# B&R Automation Studio project AAU12Segmenter (part 3)

```iecst
	(*________________________________________*)
	(*_____________KUKA5 Mappings_____________*)
	(*________________________________________*)

	::InputVariables[4,0] AT %IB."KUKA5_KRC4_ProfiNet_5_0".Module001_8_digital_inputs_I_00;
	::InputVariables[4,1] AT %IB."KUKA5_KRC4_ProfiNet_5_0".Module001_8_digital_inputs_I_01;
	::InputVariables[4,2] AT %IB."KUKA5_KRC4_ProfiNet_5_0".Module001_8_digital_inputs_I_02;
	::InputVariables[4,3] AT %IB."KUKA5_KRC4_ProfiNet_5_0".Module001_8_digital_inputs_I_03;
	::InputVariables[4,4] AT %IB."KUKA5_KRC4_ProfiNet_5_0".Module001_8_digital_inputs_I_04;
	::InputVariables[4,5] AT %IB."KUKA5_KRC4_ProfiNet_5_0".Module001_8_digital_inputs_I_05;
	::InputVariables[4,6] AT %IB."KUKA5_KRC4_ProfiNet_5_0".Module001_8_digital_inputs_I_06;
	::InputVariables[4,7] AT %IB."KUKA5_KRC4_ProfiNet_5_0".Module001_8_digital_inputs_I_07;
	::InputVariables[4,8] AT %IB."KUKA5_KRC4_ProfiNet_5_0".Module001_8_digital_inputs_I_08;
	::InputVariables[4,9] AT %IB."KUKA5_KRC4_ProfiNet_5_0".Module001_8_digital_inputs_I_09;
	::InputVariables[4,10] AT %IB."KUKA5_KRC4_ProfiNet_5_0".Module001_8_digital_inputs_I_10;
	::InputVariables[4,11] AT %IB."KUKA5_KRC4_ProfiNet_5_0".Module001_8_digital_inputs_I_11;
	::InputVariables[4,12] AT %IB."KUKA5_KRC4_ProfiNet_5_0".Module001_8_digital_inputs_I_12;
	::InputVariables[4,13] AT %IB."KUKA5_KRC4_ProfiNet_5_0".Module001_8_digital_inputs_I_13;
	::InputVariables[4,14] AT %IB."KUKA5_KRC4_ProfiNet_5_0".Module001_8_digital_inputs_I_14;
	::InputVariables[4,15] AT %IB."KUKA5_KRC4_ProfiNet_5_0".Module001_8_digital_inputs_I_15;
	::InputVariables[4,16] AT %IB."KUKA5_KRC4_ProfiNet_5_0".Module001_8_digital_inputs_I_16;
	::InputVariables[4,17] AT %IB."KUKA5_KRC4_ProfiNet_5_0".Module001_8_digital_inputs_I_17;
	::InputVariables[4,18] AT %IB."KUKA5_KRC4_ProfiNet_5_0".Module001_8_digital_inputs_I_18;
	::InputVariables[4,19] AT %IB."KUKA5_KRC4_ProfiNet_5_0".Module001_8_digital_inputs_I_19;
	::InputVariables[4,20] AT %IB."KUKA5_KRC4_ProfiNet_5_0".Module001_8_digital_inputs_I_20;
	::InputVariables[4,21] AT %IB."KUKA5_KRC4_ProfiNet_5_0".Module001_8_digital_inputs_I_21;
	::InputVariables[4,22] AT %IB."KUKA5_KRC4_ProfiNet_5_0".Module001_8_digital_inputs_I_22;
	::InputVariables[4,23] AT %IB."KUKA5_KRC4_ProfiNet_5_0".Module001_8_digital_inputs_I_23;
	::InputVariables[4,24] AT %IB."KUKA5_KRC4_ProfiNet_5_0".Module001_8_digital_inputs_I_24;
	::InputVariables[4,25] AT %IB."KUKA5_KRC4_ProfiNet_5_0".Module001_8_digital_inputs_I_25;
	::InputVariables[4,26] AT %IB."KUKA5_KRC4_ProfiNet_5_0".Module001_8_digital_inputs_I_26;
	::InputVariables[4,27] AT %IB."KUKA5_KRC4_ProfiNet_5_0".Module001_8_digital_inputs_I_27;
	::InputVariables[4,28] AT %IB."KUKA5_KRC4_ProfiNet_5_0".Module001_8_digital_inputs_I_28;
	::InputVariables[4,29] AT %IB."KUKA5_KRC4_ProfiNet_5_0".Module001_8_digital_inputs_I_29;
	::InputVariables[4,30] AT %IB."KUKA5_KRC4_ProfiNet_5_0".Module001_8_digital_inputs_I_30;
	::InputVariables[4,31] AT %IB."KUKA5_KRC4_ProfiNet_5_0".Module001_8_digital_inputs_I_31;
	::InputVariables[4,32] AT %IB."KUKA5_KRC4_ProfiNet_5_0".Module001_8_digital_inputs_I_32;
	::InputVariables[4,33] AT %IB."KUKA5_KRC4_ProfiNet_5_0".Module001_8_digital_inputs_I_33;
	::InputVariables[4,34] AT %IB."KUKA5_KRC4_ProfiNet_5_0".Module001_8_digital_inputs_I_34;
	::InputVariables[4,35] AT %IB."KUKA5_KRC4_ProfiNet_5_0".Module001_8_digital_inputs_I_35;
	::InputVariables[4,36] AT %IB."KUKA5_KRC4_ProfiNet_5_0".Module001_8_digital_inputs_I_36;
	::InputVariables[4,37] AT %IB."KUKA5_KRC4_ProfiNet_5_0".Module001_8_digital_inputs_I_37;
	::InputVariables[4,38] AT %IB."KUKA5_KRC4_ProfiNet_5_0".Module001_8_digital_inputs_I_38;
	::InputVariables[4,39] AT %IB."KUKA5_KRC4_ProfiNet_5_0".Module001_8_digital_inputs_I_39;
	::InputVariables[4,40] AT %IB."KUKA5_KRC4_ProfiNet_5_0".Module001_8_digital_inputs_I_40;
	::InputVariables[4,41] AT %IB."KUKA5_KRC4_ProfiNet_5_0".Module001_8_digital_inputs_I_41;
	::InputVariables[4,42] AT %IB."KUKA5_KRC4_ProfiNet_5_0".Module001_8_digital_inputs_I_42;
	::InputVariables[4,43] AT %IB."KUKA5_KRC4_ProfiNet_5_0".Module001_8_digital_inputs_I_43;
	::InputVariables[4,44] AT %IB."KUKA5_KRC4_ProfiNet_5_0".Module001_8_digital_inputs_I_44;
	::InputVariables[4,45] AT %IB."KUKA5_KRC4_ProfiNet_5_0".Module001_8_digital_inputs_I_45;
	::InputVariables[4,46] AT %IB."KUKA5_KRC4_ProfiNet_5_0".Module001_8_digital_inputs_I_46;
	::InputVariables[4,47] AT %IB."KUKA5_KRC4_ProfiNet_5_0".Module001_8_digital_inputs_I_47;
	::InputVariables[4,48] AT %IB."KUKA5_KRC4_ProfiNet_5_0".Module001_8_digital_inputs_I_48;
	::InputVariables[4,49] AT %IB."KUKA5_KRC4_ProfiNet_5_0".Module001_8_digital_inputs_I_49;
	::InputVariables[4,50] AT %IB."KUKA5_KRC4_ProfiNet_5_0".Module001_8_digital_inputs_I_50;
	::InputVariables[4,51] AT %IB."KUKA5_KRC4_ProfiNet_5_0".Module001_8_digital_inputs_I_51;
	::InputVariables[4,52] AT %IB."KUKA5_KRC4_ProfiNet_5_0".Module001_8_digital_inputs_I_52;
	::InputVariables[4,53] AT %IB."KUKA5_KRC4_ProfiNet_5_0".Module001_8_digital_inputs_I_53;
	::InputVariables[4,54] AT %IB."KUKA5_KRC4_ProfiNet_5_0".Module001_8_digital_inputs_I_54;
	::InputVariables[4,55] AT %IB."KUKA5_KRC4_ProfiNet_5_0".Module001_8_digital_inputs_I_55;
	::InputVariables[4,56] AT %IB."KUKA5_KRC4_ProfiNet_5_0".Module001_8_digital_inputs_I_56;
	::InputVariables[4,57] AT %IB."KUKA5_KRC4_ProfiNet_5_0".Module001_8_digital_inputs_I_57;
	::InputVariables[4,58] AT %IB."KUKA5_KRC4_ProfiNet_5_0".Module001_8_digital_inputs_I_58;
	::InputVariables[4,59] AT %IB."KUKA5_KRC4_ProfiNet_5_0".Module001_8_digital_inputs_I_59;
	::InputVariables[4,60] AT %IB."KUKA5_KRC4_ProfiNet_5_0".Module001_8_digital_inputs_I_60;
	::InputVariables[4,61] AT %IB."KUKA5_KRC4_ProfiNet_5_0".Module001_8_digital_inputs_I_61;
	::InputVariables[4,62] AT %IB."KUKA5_KRC4_ProfiNet_5_0".Module001_8_digital_inputs_I_62;
	::InputVariables[4,63] AT %IB."KUKA5_KRC4_ProfiNet_5_0".Module001_8_digital_inputs_I_63;
	::InputVariables[4,64] AT %IB."KUKA5_KRC4_ProfiNet_5_0".Module001_8_digital_inputs_I_64;
	::InputVariables[4,65] AT %IB."KUKA5_KRC4_ProfiNet_5_0".Module001_8_digital_inputs_I_65;
	::InputVariables[4,66] AT %IB."KUKA5_KRC4_ProfiNet_5_0".Module001_8_digital_inputs_I_66;
	::InputVariables[4,67] AT %IB."KUKA5_KRC4_ProfiNet_5_0".Module001_8_digital_inputs_I_67;
	::InputVariables[4,68] AT %IB."KUKA5_KRC4_ProfiNet_5_0".Module001_8_digital_inputs_I_68;
	::InputVariables[4,69] AT %IB."KUKA5_KRC4_ProfiNet_5_0".Module001_8_digital_inputs_I_69;
	::InputVariables[4,70] AT %IB."KUKA5_KRC4_ProfiNet_5_0".Module001_8_digital_inputs_I_70;
	::InputVariables[4,71] AT %IB."KUKA5_KRC4_ProfiNet_5_0".Module001_8_digital_inputs_I_71;
	::InputVariables[4,72] AT %IB."KUKA5_KRC4_ProfiNet_5_0".Module001_8_digital_inputs_I_72;
	::InputVariables[4,73] AT %IB."KUKA5_KRC4_ProfiNet_5_0".Module001_8_digital_inputs_I_73;
	::InputVariables[4,74] AT %IB."KUKA5_KRC4_ProfiNet_5_0".Module001_8_digital_inputs_I_74;
	::InputVariables[4,75] AT %IB."KUKA5_KRC4_ProfiNet_5_0".Module001_8_digital_inputs_I_75;
	::InputVariables[4,76] AT %IB."KUKA5_KRC4_ProfiNet_5_0".Module001_8_digital_inputs_I_76;
	::InputVariables[4,77] AT %IB."KUKA5_KRC4_ProfiNet_5_0".Module001_8_digital_inputs_I_77;
	::InputVariables[4,78] AT %IB."KUKA5_KRC4_ProfiNet_5_0".Module001_8_digital_inputs_I_78;
	::InputVariables[4,79] AT %IB."KUKA5_KRC4_ProfiNet_5_0".Module001_8_digital_inputs_I_79;
	::InputVariables[4,80] AT %IB."KUKA5_KRC4_ProfiNet_5_0".Module001_8_digital_inputs_I_80;
	::InputVariables[4,81] AT %IB."KUKA5_KRC4_ProfiNet_5_0".Module001_8_digital_inputs_I_81;
	::InputVariables[4,82] AT %IB."KUKA5_KRC4_ProfiNet_5_0".Module001_8_digital_inputs_I_82;
	::InputVariables[4,83] AT %IB."KUKA5_KRC4_ProfiNet_5_0".Module001_8_digital_inputs_I_83;
	::InputVariables[4,84] AT %IB."KUKA5_KRC4_ProfiNet_5_0".Module001_8_digital_inputs_I_84;
	::InputVariables[4,85] AT %IB."KUKA5_KRC4_ProfiNet_5_0".Module001_8_digital_inputs_I_85;
	::InputVariables[4,86] AT %IB."KUKA5_KRC4_ProfiNet_5_0".Module001_8_digital_inputs_I_86;
	::InputVariables[4,87] AT %IB."KUKA5_KRC4_ProfiNet_5_0".Module001_8_digital_inputs_I_87;
	::InputVariables[4,88] AT %IB."KUKA5_KRC4_ProfiNet_5_0".Module001_8_digital_inputs_I_88;
	::InputVariables[4,89] AT %IB."KUKA5_KRC4_ProfiNet_5_0".Module001_8_digital_inputs_I_89;
	::InputVariables[4,90] AT %IB."KUKA5_KRC4_ProfiNet_5_0".Module001_8_digital_inputs_I_90;
	::InputVariables[4,91] AT %IB."KUKA5_KRC4_ProfiNet_5_0".Module001_8_digital_inputs_I_91;
	::InputVariables[4,92] AT %IB."KUKA5_KRC4_ProfiNet_5_0".Module001_8_digital_inputs_I_92;
	::InputVariables[4,93] AT %IB."KUKA5_KRC4_ProfiNet_5_0".Module001_8_digital_inputs_I_93;
	::InputVariables[4,94] AT %IB."KUKA5_KRC4_ProfiNet_5_0".Module001_8_digital_inputs_I_94;
	::InputVariables[4,95] AT %IB."KUKA5_KRC4_ProfiNet_5_0".Module001_8_digital_inputs_I_95;
	::InputVariables[4,96] AT %IB."KUKA5_KRC4_ProfiNet_5_0".Module001_8_digital_inputs_I_96;
	::InputVariables[4,97] AT %IB."KUKA5_KRC4_ProfiNet_5_0".Module001_8_digital_inputs_I_97;
	::InputVariables[4,98] AT %IB."KUKA5_KRC4_ProfiNet_5_0".Module001_8_digital_inputs_I_98;
	::InputVariables[4,99] AT %IB."KUKA5_KRC4_ProfiNet_5_0".Module001_8_digital_inputs_I_99;
	::InputVariables[4,100] AT %IB."KUKA5_KRC4_ProfiNet_5_0".Module001_8_digital_inputs_I_100;
	::InputVariables[4,101] AT %IB."KUKA5_KRC4_ProfiNet_5_0".Module001_8_digital_inputs_I_101;
	::InputVariables[4,102] AT %IB."KUKA5_KRC4_ProfiNet_5_0".Module001_8_digital_inputs_I_102;
	::InputVariables[4,103] AT %IB."KUKA5_KRC4_ProfiNet_5_0".Module001_8_digital_inputs_I_103;
	::InputVariables[4,104] AT %IB."KUKA5_KRC4_ProfiNet_5_0".Module001_8_digital_inputs_I_104;
	::InputVariables[4,105] AT %IB."KUKA5_KRC4_ProfiNet_5_0".Module001_8_digital_inputs_I_105;
	::InputVariables[4,106] AT %IB."KUKA5_KRC4_ProfiNet_5_0".Module001_8_digital_inputs_I_106;
	::InputVariables[4,107] AT %IB."KUKA5_KRC4_ProfiNet_5_0".Module001_8_digital_inputs_I_107;
	::InputVariables[4,108] AT %IB."KUKA5_KRC4_ProfiNet_5_0".Module001_8_digital_inputs_I_108;
	::InputVariables[4,109] AT %IB."KUKA5_KRC4_ProfiNet_5_0".Module001_8_digital_inputs_I_109;
	::InputVariables[4,110] AT %IB."KUKA5_KRC4_ProfiNet_5_0".Module001_8_digital_inputs_I_110;
	::InputVariables[4,111] AT %IB."KUKA5_KRC4_ProfiNet_5_0".Module001_8_digital_inputs_I_111;
	::InputVariables[4,112] AT %IB."KUKA5_KRC4_ProfiNet_5_0".Module001_8_digital_inputs_I_112;
	::InputVariables[4,113] AT %IB."KUKA5_KRC4_ProfiNet_5_0".Module001_8_digital_inputs_I_113;
	::InputVariables[4,114] AT %IB."KUKA5_KRC4_ProfiNet_5_0".Module001_8_digital_inputs_I_114;
	::InputVariables[4,115] AT %IB."KUKA5_KRC4_ProfiNet_5_0".Module001_8_digital_inputs_I_115;
	::InputVariables[4,116] AT %IB."KUKA5_KRC4_ProfiNet_5_0".Module001_8_digital_inputs_I_116;
	::InputVariables[4,117] AT %IB."KUKA5_KRC4_ProfiNet_5_0".Module001_8_digital_inputs_I_117;
	::InputVariables[4,118] AT %IB."KUKA5_KRC4_ProfiNet_5_0".Module001_8_digital_inputs_I_118;
	::InputVariables[4,119] AT %IB."KUKA5_KRC4_ProfiNet_5_0".Module001_8_digital_inputs_I_119;
	::InputVariables[4,120] AT %IB."KUKA5_KRC4_ProfiNet_5_0".Module001_8_digital_inputs_I_120;
	::InputVariables[4,121] AT %IB."KUKA5_KRC4_ProfiNet_5_0".Module001_8_digital_inputs_I_121;
	::InputVariables[4,122] AT %IB."KUKA5_KRC4_ProfiNet_5_0".Module001_8_digital_inputs_I_122;
	::InputVariables[4,123] AT %IB."KUKA5_KRC4_ProfiNet_5_0".Module001_8_digital_inputs_I_123;
	::InputVariables[4,124] AT %IB."KUKA5_KRC4_ProfiNet_5_0".Module001_8_digital_inputs_I_124;
	::InputVariables[4,125] AT %IB."KUKA5_KRC4_ProfiNet_5_0".Module001_8_digital_inputs_I_125;
	::InputVariables[4,126] AT %IB."KUKA5_KRC4_ProfiNet_5_0".Module001_8_digital_inputs_I_126;
	::InputVariables[4,127] AT %IB."KUKA5_KRC4_ProfiNet_5_0".Module001_8_digital_inputs_I_127;
	::InputVariables[4,128] AT %IB."KUKA5_KRC4_ProfiNet_5_0".Module001_8_digital_inputs_I_128;
	::InputVariables[4,129] AT %IB."KUKA5_KRC4_ProfiNet_5_0".Module001_8_digital_inputs_I_129;
	::InputVariables[4,130] AT %IB."KUKA5_KRC4_ProfiNet_5_0".Module001_8_digital_inputs_I_130;
	::InputVariables[4,131] AT %IB."KUKA5_KRC4_ProfiNet_5_0".Module001_8_digital_inputs_I_131;
	::InputVariables[4,132] AT %IB."KUKA5_KRC4_ProfiNet_5_0".Module001_8_digital_inputs_I_132;
	::InputVariables[4,133] AT %IB."KUKA5_KRC4_ProfiNet_5_0".Module001_8_digital_inputs_I_133;
	::InputVariables[4,134] AT %IB."KUKA5_KRC4_ProfiNet_5_0".Module001_8_digital_inputs_I_134;
	::InputVariables[4,135] AT %IB."KUKA5_KRC4_ProfiNet_5_0".Module001_8_digital_inputs_I_135;
	::InputVariables[4,136] AT %IB."KUKA5_KRC4_ProfiNet_5_0".Module001_8_digital_inputs_I_136;
	::InputVariables[4,137] AT %IB."KUKA5_KRC4_ProfiNet_5_0".Module001_8_digital_inputs_I_137;
	::InputVariables[4,138] AT %IB."KUKA5_KRC4_ProfiNet_5_0".Module001_8_digital_inputs_I_138;
	::InputVariables[4,139] AT %IB."KUKA5_KRC4_ProfiNet_5_0".Module001_8_digital_inputs_I_139;
	::InputVariables[4,140] AT %IB."KUKA5_KRC4_ProfiNet_5_0".Module001_8_digital_inputs_I_140;
	::InputVariables[4,141] AT %IB."KUKA5_KRC4_ProfiNet_5_0".Module001_8_digital_inputs_I_141;
	::InputVariables[4,142] AT %IB."KUKA5_KRC4_ProfiNet_5_0".Module001_8_digital_inputs_I_142;
	::InputVariables[4,143] AT %IB."KUKA5_KRC4_ProfiNet_5_0".Module001_8_digital_inputs_I_143;
	::InputVariables[4,144] AT %IB."KUKA5_KRC4_ProfiNet_5_0".Module001_8_digital_inputs_I_144;
	::InputVariables[4,145] AT %IB."KUKA5_KRC4_ProfiNet_5_0".Module001_8_digital_inputs_I_145;
	::InputVariables[4,146] AT %IB."KUKA5_KRC4_ProfiNet_5_0".Module001_8_digital_inputs_I_146;
	::InputVariables[4,147] AT %IB."KUKA5_KRC4_ProfiNet_5_0".Module001_8_digital_inputs_I_147;
	::InputVariables[4,148] AT %IB."KUKA5_KRC4_ProfiNet_5_0".Module001_8_digital_inputs_I_148;
	::InputVariables[4,149] AT %IB."KUKA5_KRC4_ProfiNet_5_0".Module001_8_digital_inputs_I_149;
	::InputVariables[4,150] AT %IB."KUKA5_KRC4_ProfiNet_5_0".Module001_8_digital_inputs_I_150;
	::InputVariables[4,151] AT %IB."KUKA5_KRC4_ProfiNet_5_0".Module001_8_digital_inputs_I_151;
	::InputVariables[4,152] AT %IB."KUKA5_KRC4_ProfiNet_5_0".Module001_8_digital_inputs_I_152;
	::InputVariables[4,153] AT %IB."KUKA5_KRC4_ProfiNet_5_0".Module001_8_digital_inputs_I_153;
	::InputVariables[4,154] AT %IB."KUKA5_KRC4_ProfiNet_5_0".Module001_8_digital_inputs_I_154;
	::InputVariables[4,155] AT %IB."KUKA5_KRC4_ProfiNet_5_0".Module001_8_digital_inputs_I_155;
	::InputVariables[4,156] AT %IB."KUKA5_KRC4_ProfiNet_5_0".Module001_8_digital_inputs_I_156;
	::InputVariables[4,157] AT %IB."KUKA5_KRC4_ProfiNet_5_0".Module001_8_digital_inputs_I_157;
	::InputVariables[4,158] AT %IB."KUKA5_KRC4_ProfiNet_5_0".Module001_8_digital_inputs_I_158;
	::InputVariables[4,159] AT %IB."KUKA5_KRC4_ProfiNet_5_0".Module001_8_digital_inputs_I_159;
	::InputVariables[4,160] AT %IB."KUKA5_KRC4_ProfiNet_5_0".Module001_8_digital_inputs_I_160;
	::InputVariables[4,161] AT %IB."KUKA5_KRC4_ProfiNet_5_0".Module001_8_digital_inputs_I_161;
	::InputVariables[4,162] AT %IB."KUKA5_KRC4_ProfiNet_5_0".Module001_8_digital_inputs_I_162;
	::InputVariables[4,163] AT %IB."KUKA5_KRC4_ProfiNet_5_0".Module001_8_digital_inputs_I_163;
	::InputVariables[4,164] AT %IB."KUKA5_KRC4_ProfiNet_5_0".Module001_8_digital_inputs_I_164;
	::InputVariables[4,165] AT %IB."KUKA5_KRC4_ProfiNet_5_0".Module001_8_digital_inputs_I_165;
	::InputVariables[4,166] AT %IB."KUKA5_KRC4_ProfiNet_5_0".Module001_8_digital_inputs_I_166;
	::InputVariables[4,167] AT %IB."KUKA5_KRC4_ProfiNet_5_0".Module001_8_digital_inputs_I_167;
	::InputVariables[4,168] AT %IB."KUKA5_KRC4_ProfiNet_5_0".Module001_8_digital_inputs_I_168;
	::InputVariables[4,169] AT %IB."KUKA5_KRC4_ProfiNet_5_0".Module001_8_digital_inputs_I_169;
	::InputVariables[4,170] AT %IB."KUKA5_KRC4_ProfiNet_5_0".Module001_8_digital_inputs_I_170;
	::InputVariables[4,171] AT %IB."KUKA5_KRC4_ProfiNet_5_0".Module001_8_digital_inputs_I_171;
	::InputVariables[4,172] AT %IB."KUKA5_KRC4_ProfiNet_5_0".Module001_8_digital_inputs_I_172;
	::InputVariables[4,173] AT %IB."KUKA5_KRC4_ProfiNet_5_0".Module001_8_digital_inputs_I_173;
	::InputVariables[4,174] AT %IB."KUKA5_KRC4_ProfiNet_5_0".Module001_8_digital_inputs_I_174;
	::InputVariables[4,175] AT %IB."KUKA5_KRC4_ProfiNet_5_0".Module001_8_digital_inputs_I_175;
	::InputVariables[4,176] AT %IB."KUKA5_KRC4_ProfiNet_5_0".Module001_8_digital_inputs_I_176;
	::InputVariables[4,177] AT %IB."KUKA5_KRC4_ProfiNet_5_0".Module001_8_digital_inputs_I_177;
	::InputVariables[4,178] AT %IB."KUKA5_KRC4_ProfiNet_5_0".Module001_8_digital_inputs_I_178;
	::InputVariables[4,179] AT %IB."KUKA5_KRC4_ProfiNet_5_0".Module001_8_digital_inputs_I_179;
	::InputVariables[4,180] AT %IB."KUKA5_KRC4_ProfiNet_5_0".Module001_8_digital_inputs_I_180;
	::InputVariables[4,181] AT %IB."KUKA5_KRC4_ProfiNet_5_0".Module001_8_digital_inputs_I_181;
	::InputVariables[4,182] AT %IB."KUKA5_KRC4_ProfiNet_5_0".Module001_8_digital_inputs_I_182;
	::InputVariables[4,183] AT %IB."KUKA5_KRC4_ProfiNet_5_0".Module001_8_digital_inputs_I_183;
	::InputVariables[4,184] AT %IB."KUKA5_KRC4_ProfiNet_5_0".Module001_8_digital_inputs_I_184;
	::InputVariables[4,185] AT %IB."KUKA5_KRC4_ProfiNet_5_0".Module001_8_digital_inputs_I_185;
	::InputVariables[4,186] AT %IB."KUKA5_KRC4_ProfiNet_5_0".Module001_8_digital_inputs_I_186;
	::InputVariables[4,187] AT %IB."KUKA5_KRC4_ProfiNet_5_0".Module001_8_digital_inputs_I_187;
	::InputVariables[4,188] AT %IB."KUKA5_KRC4_ProfiNet_5_0".Module001_8_digital_inputs_I_188;
	::InputVariables[4,189] AT %IB."KUKA5_KRC4_ProfiNet_5_0".Module001_8_digital_inputs_I_189;
	::InputVariables[4,190] AT %IB."KUKA5_KRC4_ProfiNet_5_0".Module001_8_digital_inputs_I_190;
	::InputVariables[4,191] AT %IB."KUKA5_KRC4_ProfiNet_5_0".Module001_8_digital_inputs_I_191;
	::InputVariables[4,192] AT %IB."KUKA5_KRC4_ProfiNet_5_0".Module001_8_digital_inputs_I_192;
	::InputVariables[4,193] AT %IB."KUKA5_KRC4_ProfiNet_5_0".Module001_8_digital_inputs_I_193;
	::InputVariables[4,194] AT %IB."KUKA5_KRC4_ProfiNet_5_0".Module001_8_digital_inputs_I_194;
	::InputVariables[4,195] AT %IB."KUKA5_KRC4_ProfiNet_5_0".Module001_8_digital_inputs_I_195;
	::InputVariables[4,196] AT %IB."KUKA5_KRC4_ProfiNet_5_0".Module001_8_digital_inputs_I_196;
	::InputVariables[4,197] AT %IB."KUKA5_KRC4_ProfiNet_5_0".Module001_8_digital_inputs_I_197;
	::InputVariables[4,198] AT %IB."KUKA5_KRC4_ProfiNet_5_0".Module001_8_digital_inputs_I_198;
	::InputVariables[4,199] AT %IB."KUKA5_KRC4_ProfiNet_5_0".Module001_8_digital_inputs_I_199;
	::InputVariables[4,200] AT %IB."KUKA5_KRC4_ProfiNet_5_0".Module001_8_digital_inputs_I_200;
	::InputVariables[4,201] AT %IB."KUKA5_KRC4_ProfiNet_5_0".Module001_8_digital_inputs_I_201;
	::InputVariables[4,202] AT %IB."KUKA5_KRC4_ProfiNet_5_0".Module001_8_digital_inputs_I_202;
	::InputVariables[4,203] AT %IB."KUKA5_KRC4_ProfiNet_5_0".Module001_8_digital_inputs_I_203;
	::InputVariables[4,204] AT %IB."KUKA5_KRC4_ProfiNet_5_0".Module001_8_digital_inputs_I_204;
	::InputVariables[4,205] AT %IB."KUKA5_KRC4_ProfiNet_5_0".Module001_8_digital_inputs_I_205;
	::InputVariables[4,206] AT %IB."KUKA5_KRC4_ProfiNet_5_0".Module001_8_digital_inputs_I_206;
	::InputVariables[4,207] AT %IB."KUKA5_KRC4_ProfiNet_5_0".Module001_8_digital_inputs_I_207;
	::InputVariables[4,208] AT %IB."KUKA5_KRC4_ProfiNet_5_0".Module001_8_digital_inputs_I_208;
	::InputVariables[4,209] AT %IB."KUKA5_KRC4_ProfiNet_5_0".Module001_8_digital_inputs_I_209;
	::InputVariables[4,210] AT %IB."KUKA5_KRC4_ProfiNet_5_0".Module001_8_digital_inputs_I_210;
	::InputVariables[4,211] AT %IB."KUKA5_KRC4_ProfiNet_5_0".Module001_8_digital_inputs_I_211;
	::InputVariables[4,212] AT %IB."KUKA5_KRC4_ProfiNet_5_0".Module001_8_digital_inputs_I_212;
	::InputVariables[4,213] AT %IB."KUKA5_KRC4_ProfiNet_5_0".Module001_8_digital_inputs_I_213;
	::InputVariables[4,214] AT %IB."KUKA5_KRC4_ProfiNet_5_0".Module001_8_digital_inputs_I_214;
	::InputVariables[4,215] AT %IB."KUKA5_KRC4_ProfiNet_5_0".Module001_8_digital_inputs_I_215;
	::InputVariables[4,216] AT %IB."KUKA5_KRC4_ProfiNet_5_0".Module001_8_digital_inputs_I_216;
	::InputVariables[4,217] AT %IB."KUKA5_KRC4_ProfiNet_5_0".Module001_8_digital_inputs_I_217;
	::InputVariables[4,218] AT %IB."KUKA5_KRC4_ProfiNet_5_0".Module001_8_digital_inputs_I_218;
	::InputVariables[4,219] AT %IB."KUKA5_KRC4_ProfiNet_5_0".Module001_8_digital_inputs_I_219;
	::InputVariables[4,220] AT %IB."KUKA5_KRC4_ProfiNet_5_0".Module001_8_digital_inputs_I_220;
	::InputVariables[4,221] AT %IB."KUKA5_KRC4_ProfiNet_5_0".Module001_8_digital_inputs_I_221;
	::InputVariables[4,222] AT %IB."KUKA5_KRC4_ProfiNet_5_0".Module001_8_digital_inputs_I_222;
	::InputVariables[4,223] AT %IB."KUKA5_KRC4_ProfiNet_5_0".Module001_8_digital_inputs_I_223;
	::InputVariables[4,224] AT %IB."KUKA5_KRC4_ProfiNet_5_0".Module001_8_digital_inputs_I_224;
	::InputVariables[4,225] AT %IB."KUKA5_KRC4_ProfiNet_5_0".Module001_8_digital_inputs_I_225;
	::InputVariables[4,226] AT %IB."KUKA5_KRC4_ProfiNet_5_0".Module001_8_digital_inputs_I_226;
	::InputVariables[4,227] AT %IB."KUKA5_KRC4_ProfiNet_5_0".Module001_8_digital_inputs_I_227;
	::InputVariables[4,228] AT %IB."KUKA5_KRC4_ProfiNet_5_0".Module001_8_digital_inputs_I_228;
	::InputVariables[4,229] AT %IB."KUKA5_KRC4_ProfiNet_5_0".Module001_8_digital_inputs_I_229;
	::InputVariables[4,230] AT %IB."KUKA5_KRC4_ProfiNet_5_0".Module001_8_digital_inputs_I_230;
	::InputVariables[4,231] AT %IB."KUKA5_KRC4_ProfiNet_5_0".Module001_8_digital_inputs_I_231;
	::InputVariables[4,232] AT %IB."KUKA5_KRC4_ProfiNet_5_0".Module001_8_digital_inputs_I_232;
	::InputVariables[4,233] AT %IB."KUKA5_KRC4_ProfiNet_5_0".Module001_8_digital_inputs_I_233;
	::InputVariables[4,234] AT %IB."KUKA5_KRC4_ProfiNet_5_0".Module001_8_digital_inputs_I_234;
	::InputVariables[4,235] AT %IB."KUKA5_KRC4_ProfiNet_5_0".Module001_8_digital_inputs_I_235;
	::InputVariables[4,236] AT %IB."KUKA5_KRC4_ProfiNet_5_0".Module001_8_digital_inputs_I_236;
	::InputVariables[4,237] AT %IB."KUKA5_KRC4_ProfiNet_5_0".Module001_8_digital_inputs_I_237;
	::InputVariables[4,238] AT %IB."KUKA5_KRC4_ProfiNet_5_0".Module001_8_digital_inputs_I_238;
	::InputVariables[4,239] AT %IB."KUKA5_KRC4_ProfiNet_5_0".Module001_8_digital_inputs_I_239;
	::InputVariables[4,240] AT %IB."KUKA5_KRC4_ProfiNet_5_0".Module001_8_digital_inputs_I_240;
	::InputVariables[4,241] AT %IB."KUKA5_KRC4_ProfiNet_5_0".Module001_8_digital_inputs_I_241;
	::InputVariables[4,242] AT %IB."KUKA5_KRC4_ProfiNet_5_0".Module001_8_digital_inputs_I_242;
	::InputVariables[4,243] AT %IB."KUKA5_KRC4_ProfiNet_5_0".Module001_8_digital_inputs_I_243;
	::InputVariables[4,244] AT %IB."KUKA5_KRC4_ProfiNet_5_0".Module001_8_digital_inputs_I_244;
	::InputVariables[4,245] AT %IB."KUKA5_KRC4_ProfiNet_5_0".Module001_8_digital_inputs_I_245;
	::InputVariables[4,246] AT %IB."KUKA5_KRC4_ProfiNet_5_0".Module001_8_digital_inputs_I_246;
	::InputVariables[4,247] AT %IB."KUKA5_KRC4_ProfiNet_5_0".Module001_8_digital_inputs_I_247;
	::InputVariables[4,248] AT %IB."KUKA5_KRC4_ProfiNet_5_0".Module001_8_digital_inputs_I_248;
	::InputVariables[4,249] AT %IB."KUKA5_KRC4_ProfiNet_5_0".Module001_8_digital_inputs_I_249;
	::InputVariables[4,250] AT %IB."KUKA5_KRC4_ProfiNet_5_0".Module001_8_digital_inputs_I_250;
	::InputVariables[4,251] AT %IB."KUKA5_KRC4_ProfiNet_5_0".Module001_8_digital_inputs_I_251;
	::InputVariables[4,252] AT %IB."KUKA5_KRC4_ProfiNet_5_0".Module001_8_digital_inputs_I_252;
	::InputVariables[4,253] AT %IB."KUKA5_KRC4_ProfiNet_5_0".Module001_8_digital_inputs_I_253;

	::OutputVariables[4,0]	AT %QB."KUKA5_KRC4_ProfiNet_5_0".Module001_8_digital_outputs_O_00;
	::OutputVariables[4,1]	AT %QB."KUKA5_KRC4_ProfiNet_5_0".Module001_8_digital_outputs_O_01;
	::OutputVariables[4,2]	AT %QB."KUKA5_KRC4_ProfiNet_5_0".Module001_8_digital_outputs_O_02;
	::OutputVariables[4,3]	AT %QB."KUKA5_KRC4_ProfiNet_5_0".Module001_8_digital_outputs_O_03;
	::OutputVariables[4,4]	AT %QB."KUKA5_KRC4_ProfiNet_5_0".Module001_8_digital_outputs_O_04;
	::OutputVariables[4,5]	AT %QB."KUKA5_KRC4_ProfiNet_5_0".Module001_8_digital_outputs_O_05;
	::OutputVariables[4,6]	AT %QB."KUKA5_KRC4_ProfiNet_5_0".Module001_8_digital_outputs_O_06;
	::OutputVariables[4,7]	AT %QB."KUKA5_KRC4_ProfiNet_5_0".Module001_8_digital_outputs_O_07;
	::OutputVariables[4,8]	AT %QB."KUKA5_KRC4_ProfiNet_5_0".Module001_8_digital_outputs_O_08;
	::OutputVariables[4,9]	AT %QB."KUKA5_KRC4_ProfiNet_5_0".Module001_8_digital_outputs_O_09;
	::OutputVariables[4,10]	AT %QB."KUKA5_KRC4_ProfiNet_5_0".Module001_8_digital_outputs_O_10;
	::OutputVariables[4,11]	AT %QB."KUKA5_KRC4_ProfiNet_5_0".Module001_8_digital_outputs_O_11;
	::OutputVariables[4,12]	AT %QB."KUKA5_KRC4_ProfiNet_5_0".Module001_8_digital_outputs_O_12;
	::OutputVariables[4,13]	AT %QB."KUKA5_KRC4_ProfiNet_5_0".Module001_8_digital_outputs_O_13;
	::OutputVariables[4,14]	AT %QB."KUKA5_KRC4_ProfiNet_5_0".Module001_8_digital_outputs_O_14;
	::OutputVariables[4,15]	AT %QB."KUKA5_KRC4_ProfiNet_5_0".Module001_8_digital_outputs_O_15;
	::OutputVariables[4,16]	AT %QB."KUKA5_KRC4_ProfiNet_5_0".Module001_8_digital_outputs_O_16;
	::OutputVariables[4,17]	AT %QB."KUKA5_KRC4_ProfiNet_5_0".Module001_8_digital_outputs_O_17;
	::OutputVariables[4,18]	AT %QB."KUKA5_KRC4_ProfiNet_5_0".Module001_8_digital_outputs_O_18;
	::OutputVariables[4,19]	AT %QB."KUKA5_KRC4_ProfiNet_5_0".Module001_8_digital_outputs_O_19;
	::OutputVariables[4,20]	AT %QB."KUKA5_KRC4_ProfiNet_5_0".Module001_8_digital_outputs_O_20;
	::OutputVariables[4,21]	AT %QB."KUKA5_KRC4_ProfiNet_5_0".Module001_8_digital_outputs_O_21;
	::OutputVariables[4,22]	AT %QB."KUKA5_KRC4_ProfiNet_5_0".Module001_8_digital_outputs_O_22;
	::OutputVariables[4,23]	AT %QB."KUKA5_KRC4_ProfiNet_5_0".Module001_8_digital_outputs_O_23;
	::OutputVariables[4,24]	AT %QB."KUKA5_KRC4_ProfiNet_5_0".Module001_8_digital_outputs_O_24;
	::OutputVariables[4,25]	AT %QB."KUKA5_KRC4_ProfiNet_5_0".Module001_8_digital_outputs_O_25;
	::OutputVariables[4,26]	AT %QB."KUKA5_KRC4_ProfiNet_5_0".Module001_8_digital_outputs_O_26;
	::OutputVariables[4,27]	AT %QB."KUKA5_KRC4_ProfiNet_5_0".Module001_8_digital_outputs_O_27;
	::OutputVariables[4,28]	AT %QB."KUKA5_KRC4_ProfiNet_5_0".Module001_8_digital_outputs_O_28;
	::OutputVariables[4,29]	AT %QB."KUKA5_KRC4_ProfiNet_5_0".Module001_8_digital_outputs_O_29;
	::OutputVariables[4,30]	AT %QB."KUKA5_KRC4_ProfiNet_5_0".Module001_8_digital_outputs_O_30;
	::OutputVariables[4,31]	AT %QB."KUKA5_KRC4_ProfiNet_5_0".Module001_8_digital_outputs_O_31;
	::OutputVariables[4,32]	AT %QB."KUKA5_KRC4_ProfiNet_5_0".Module001_8_digital_outputs_O_32;
	::OutputVariables[4,33]	AT %QB."KUKA5_KRC4_ProfiNet_5_0".Module001_8_digital_outputs_O_33;
	::OutputVariables[4,34]	AT %QB."KUKA5_KRC4_ProfiNet_5_0".Module001_8_digital_outputs_O_34;
	::OutputVariables[4,35]	AT %QB."KUKA5_KRC4_ProfiNet_5_0".Module001_8_digital_outputs_O_35;
	::OutputVariables[4,36]	AT %QB."KUKA5_KRC4_ProfiNet_5_0".Module001_8_digital_outputs_O_36;
	::OutputVariables[4,37]	AT %QB."KUKA5_KRC4_ProfiNet_5_0".Module001_8_digital_outputs_O_37;
	::OutputVariables[4,38]	AT %QB."KUKA5_KRC4_ProfiNet_5_0".Module001_8_digital_outputs_O_38;
	::OutputVariables[4,39]	AT %QB."KUKA5_KRC4_ProfiNet_5_0".Module001_8_digital_outputs_O_39;
	::OutputVariables[4,40]	AT %QB."KUKA5_KRC4_ProfiNet_5_0".Module001_8_digital_outputs_O_40;
	::OutputVariables[4,41]	AT %QB."KUKA5_KRC4_ProfiNet_5_0".Module001_8_digital_outputs_O_41;
	::OutputVariables[4,42]	AT %QB."KUKA5_KRC4_ProfiNet_5_0".Module001_8_digital_outputs_O_42;
	::OutputVariables[4,43]	AT %QB."KUKA5_KRC4_ProfiNet_5_0".Module001_8_digital_outputs_O_43;
	::OutputVariables[4,44]	AT %QB."KUKA5_KRC4_ProfiNet_5_0".Module001_8_digital_outputs_O_44;
	::OutputVariables[4,45]	AT %QB."KUKA5_KRC4_ProfiNet_5_0".Module001_8_digital_outputs_O_45;
	::OutputVariables[4,46]	AT %QB."KUKA5_KRC4_ProfiNet_5_0".Module001_8_digital_outputs_O_46;
	::OutputVariables[4,47]	AT %QB."KUKA5_KRC4_ProfiNet_5_0".Module001_8_digital_outputs_O_47;
	::OutputVariables[4,48]	AT %QB."KUKA5_KRC4_ProfiNet_5_0".Module001_8_digital_outputs_O_48;
	::OutputVariables[4,49]	AT %QB."KUKA5_KRC4_ProfiNet_5_0".Module001_8_digital_outputs_O_49;
	::OutputVariables[4,50]	AT %QB."KUKA5_KRC4_ProfiNet_5_0".Module001_8_digital_outputs_O_50;
	::OutputVariables[4,51]	AT %QB."KUKA5_KRC4_ProfiNet_5_0".Module001_8_digital_outputs_O_51;
	::OutputVariables[4,52]	AT %QB."KUKA5_KRC4_ProfiNet_5_0".Module001_8_digital_outputs_O_52;
	::OutputVariables[4,53]	AT %QB."KUKA5_KRC4_ProfiNet_5_0".Module001_8_digital_outputs_O_53;
	::OutputVariables[4,54]	AT %QB."KUKA5_KRC4_ProfiNet_5_0".Module001_8_digital_outputs_O_54;
	::OutputVariables[4,55]	AT %QB."KUKA5_KRC4_ProfiNet_5_0".Module001_8_digital_outputs_O_55;
	::OutputVariables[4,56]	AT %QB."KUKA5_KRC4_ProfiNet_5_0".Module001_8_digital_outputs_O_56;
	::OutputVariables[4,57]	AT %QB."KUKA5_KRC4_ProfiNet_5_0".Module001_8_digital_outputs_O_57;
	::OutputVariables[4,58]	AT %QB."KUKA5_KRC4_ProfiNet_5_0".Module001_8_digital_outputs_O_58;
	::OutputVariables[4,59]	AT %QB."KUKA5_KRC4_ProfiNet_5_0".Module001_8_digital_outputs_O_59;
	::OutputVariables[4,60]	AT %QB."KUKA5_KRC4_ProfiNet_5_0".Module001_8_digital_outputs_O_60;
	::OutputVariables[4,61]	AT %QB."KUKA5_KRC4_ProfiNet_5_0".Module001_8_digital_outputs_O_61;
	::OutputVariables[4,62]	AT %QB."KUKA5_KRC4_ProfiNet_5_0".Module001_8_digital_outputs_O_62;
	::OutputVariables[4,63]	AT %QB."KUKA5_KRC4_ProfiNet_5_0".Module001_8_digital_outputs_O_63;
	::OutputVariables[4,64]	AT %QB."KUKA5_KRC4_ProfiNet_5_0".Module001_8_digital_outputs_O_64;
	::OutputVariables[4,65]	AT %QB."KUKA5_KRC4_ProfiNet_5_0".Module001_8_digital_outputs_O_65;
	::OutputVariables[4,66]	AT %QB."KUKA5_KRC4_ProfiNet_5_0".Module001_8_digital_outputs_O_66;
	::OutputVariables[4,67]	AT %QB."KUKA5_KRC4_ProfiNet_5_0".Module001_8_digital_outputs_O_67;
	::OutputVariables[4,68]	AT %QB."KUKA5_KRC4_ProfiNet_5_0".Module001_8_digital_outputs_O_68;
	::OutputVariables[4,69]	AT %QB."KUKA5_KRC4_ProfiNet_5_0".Module001_8_digital_outputs_O_69;
	::OutputVariables[4,70]	AT %QB."KUKA5_KRC4_ProfiNet_5_0".Module001_8_digital_outputs_O_70;
	::OutputVariables[4,71]	AT %QB."KUKA5_KRC4_ProfiNet_5_0".Module001_8_digital_outputs_O_71;
	::OutputVariables[4,72]	AT %QB."KUKA5_KRC4_ProfiNet_5_0".Module001_8_digital_outputs_O_72;
	::OutputVariables[4,73]	AT %QB."KUKA5_KRC4_ProfiNet_5_0".Module001_8_digital_outputs_O_73;
	::OutputVariables[4,74]	AT %QB."KUKA5_KRC4_ProfiNet_5_0".Module001_8_digital_outputs_O_74;
	::OutputVariables[4,75]	AT %QB."KUKA5_KRC4_ProfiNet_5_0".Module001_8_digital_outputs_O_75;
	::OutputVariables[4,76]	AT %QB."KUKA5_KRC4_ProfiNet_5_0".Module001_8_digital_outputs_O_76;
	::OutputVariables[4,77]	AT %QB."KUKA5_KRC4_ProfiNet_5_0".Module001_8_digital_outputs_O_77;
	::OutputVariables[4,78]	AT %QB."KUKA5_KRC4_ProfiNet_5_0".Module001_8_digital_outputs_O_78;
	::OutputVariables[4,79]	AT %QB."KUKA5_KRC4_ProfiNet_5_0".Module001_8_digital_outputs_O_79;
	::OutputVariables[4,80]	AT %QB."KUKA5_KRC4_ProfiNet_5_0".Module001_8_digital_outputs_O_80;
	::OutputVariables[4,81]	AT %QB."KUKA5_KRC4_ProfiNet_5_0".Module001_8_digital_outputs_O_81;
	::OutputVariables[4,82]	AT %QB."KUKA5_KRC4_ProfiNet_5_0".Module001_8_digital_outputs_O_82;
	::OutputVariables[4,83]	AT %QB."KUKA5_KRC4_ProfiNet_5_0".Module001_8_digital_outputs_O_83;
	::OutputVariables[4,84]	AT %QB."KUKA5_KRC4_ProfiNet_5_0".Module001_8_digital_outputs_O_84;
	::OutputVariables[4,85]	AT %QB."KUKA5_KRC4_ProfiNet_5_0".Module001_8_digital_outputs_O_85;
	::OutputVariables[4,86]	AT %QB."KUKA5_KRC4_ProfiNet_5_0".Module001_8_digital_outputs_O_86;
	::OutputVariables[4,87]	AT %QB."KUKA5_KRC4_ProfiNet_5_0".Module001_8_digital_outputs_O_87;
	::OutputVariables[4,88]	AT %QB."KUKA5_KRC4_ProfiNet_5_0".Module001_8_digital_outputs_O_88;
	::OutputVariables[4,89]	AT %QB."KUKA5_KRC4_ProfiNet_5_0".Module001_8_digital_outputs_O_89;
	::OutputVariables[4,90]	AT %QB."KUKA5_KRC4_ProfiNet_5_0".Module001_8_digital_outputs_O_90;
	::OutputVariables[4,91]	AT %QB."KUKA5_KRC4_ProfiNet_5_0".Module001_8_digital_outputs_O_91;
	::OutputVariables[4,92]	AT %QB."KUKA5_KRC4_ProfiNet_5_0".Module001_8_digital_outputs_O_92;
	::OutputVariables[4,93]	AT %QB."KUKA5_KRC4_ProfiNet_5_0".Module001_8_digital_outputs_O_93;
	::OutputVariables[4,94]	AT %QB."KUKA5_KRC4_ProfiNet_5_0".Module001_8_digital_outputs_O_94;
	::OutputVariables[4,95]	AT %QB."KUKA5_KRC4_ProfiNet_5_0".Module001_8_digital_outputs_O_95;
	::OutputVariables[4,96]	AT %QB."KUKA5_KRC4_ProfiNet_5_0".Module001_8_digital_outputs_O_96;
	::OutputVariables[4,97]	AT %QB."KUKA5_KRC4_ProfiNet_5_0".Module001_8_digital_outputs_O_97;
	::OutputVariables[4,98]	AT %QB."KUKA5_KRC4_ProfiNet_5_0".Module001_8_digital_outputs_O_98;
	::OutputVariables[4,99]	AT %QB."KUKA5_KRC4_ProfiNet_5_0".Module001_8_digital_outputs_O_99;
	::OutputVariables[4,100]	AT %QB."KUKA5_KRC4_ProfiNet_5_0".Module001_8_digital_outputs_O_100;
	::OutputVariables[4,101]	AT %QB."KUKA5_KRC4_ProfiNet_5_0".Module001_8_digital_outputs_O_101;
	::OutputVariables[4,102]	AT %QB."KUKA5_KRC4_ProfiNet_5_0".Module001_8_digital_outputs_O_102;
	::OutputVariables[4,103]	AT %QB."KUKA5_KRC4_ProfiNet_5_0".Module001_8_digital_outputs_O_103;
	::OutputVariables[4,104]	AT %QB."KUKA5_KRC4_ProfiNet_5_0".Module001_8_digital_outputs_O_104;
	::OutputVariables[4,105]	AT %QB."KUKA5_KRC4_ProfiNet_5_0".Module001_8_digital_outputs_O_105;
	::OutputVariables[4,106]	AT %QB."KUKA5_KRC4_ProfiNet_5_0".Module001_8_digital_outputs_O_106;
	::OutputVariables[4,107]	AT %QB."KUKA5_KRC4_ProfiNet_5_0".Module001_8_digital_outputs_O_107;
	::OutputVariables[4,108]	AT %QB."KUKA5_KRC4_ProfiNet_5_0".Module001_8_digital_outputs_O_108;
	::OutputVariables[4,109]	AT %QB."KUKA5_KRC4_ProfiNet_5_0".Module001_8_digital_outputs_O_109;
	::OutputVariables[4,110]	AT %QB."KUKA5_KRC4_ProfiNet_5_0".Module001_8_digital_outputs_O_110;
	::OutputVariables[4,111]	AT %QB."KUKA5_KRC4_ProfiNet_5_0".Module001_8_digital_outputs_O_111;
	::OutputVariables[4,112]	AT %QB."KUKA5_KRC4_ProfiNet_5_0".Module001_8_digital_outputs_O_112;
	::OutputVariables[4,113]	AT %QB."KUKA5_KRC4_ProfiNet_5_0".Module001_8_digital_outputs_O_113;
	::OutputVariables[4,114]	AT %QB."KUKA5_KRC4_ProfiNet_5_0".Module001_8_digital_outputs_O_114;
	::OutputVariables[4,115]	AT %QB."KUKA5_KRC4_ProfiNet_5_0".Module001_8_digital_outputs_O_115;
	::OutputVariables[4,116]	AT %QB."KUKA5_KRC4_ProfiNet_5_0".Module001_8_digital_outputs_O_116;
	::OutputVariables[4,117]	AT %QB."KUKA5_KRC4_ProfiNet_5_0".Module001_8_digital_outputs_O_117;
	::OutputVariables[4,118]	AT %QB."KUKA5_KRC4_ProfiNet_5_0".Module001_8_digital_outputs_O_118;
	::OutputVariables[4,119]	AT %QB."KUKA5_KRC4_ProfiNet_5_0".Module001_8_digital_outputs_O_119;
	::OutputVariables[4,120]	AT %QB."KUKA5_KRC4_ProfiNet_5_0".Module001_8_digital_outputs_O_120;
	::OutputVariables[4,121]	AT %QB."KUKA5_KRC4_ProfiNet_5_0".Module001_8_digital_outputs_O_121;
	::OutputVariables[4,122]	AT %QB."KUKA5_KRC4_ProfiNet_5_0".Module001_8_digital_outputs_O_122;
	::OutputVariables[4,123]	AT %QB."KUKA5_KRC4_ProfiNet_5_0".Module001_8_digital_outputs_O_123;
	::OutputVariables[4,124]	AT %QB."KUKA5_KRC4_ProfiNet_5_0".Module001_8_digital_outputs_O_124;
	::OutputVariables[4,125]	AT %QB."KUKA5_KRC4_ProfiNet_5_0".Module001_8_digital_outputs_O_125;
	::OutputVariables[4,126]	AT %QB."KUKA5_KRC4_ProfiNet_5_0".Module001_8_digital_outputs_O_126;
	::OutputVariables[4,127]	AT %QB."KUKA5_KRC4_ProfiNet_5_0".Module001_8_digital_outputs_O_127;
	::OutputVariables[4,128]	AT %QB."KUKA5_KRC4_ProfiNet_5_0".Module001_8_digital_outputs_O_128;
	::OutputVariables[4,129]	AT %QB."KUKA5_KRC4_ProfiNet_5_0".Module001_8_digital_outputs_O_129;
	::OutputVariables[4,130]	AT %QB."KUKA5_KRC4_ProfiNet_5_0".Module001_8_digital_outputs_O_130;
	::OutputVariables[4,131]	AT %QB."KUKA5_KRC4_ProfiNet_5_0".Module001_8_digital_outputs_O_131;
	::OutputVariables[4,132]	AT %QB."KUKA5_KRC4_ProfiNet_5_0".Module001_8_digital_outputs_O_132;
	::OutputVariables[4,133]	AT %QB."KUKA5_KRC4_ProfiNet_5_0".Module001_8_digital_outputs_O_133;
	::OutputVariables[4,134]	AT %QB."KUKA5_KRC4_ProfiNet_5_0".Module001_8_digital_outputs_O_134;
	::OutputVariables[4,135]	AT %QB."KUKA5_KRC4_ProfiNet_5_0".Module001_8_digital_outputs_O_135;
	::OutputVariables[4,136]	AT %QB."KUKA5_KRC4_ProfiNet_5_0".Module001_8_digital_outputs_O_136;
	::OutputVariables[4,137]	AT %QB."KUKA5_KRC4_ProfiNet_5_0".Module001_8_digital_outputs_O_137;
	::OutputVariables[4,138]	AT %QB."KUKA5_KRC4_ProfiNet_5_0".Module001_8_digital_outputs_O_138;
	::OutputVariables[4,139]	AT %QB."KUKA5_KRC4_ProfiNet_5_0".Module001_8_digital_outputs_O_139;
	::OutputVariables[4,140]	AT %QB."KUKA5_KRC4_ProfiNet_5_0".Module001_8_digital_outputs_O_140;
	::OutputVariables[4,141]	AT %QB."KUKA5_KRC4_ProfiNet_5_0".Module001_8_digital_outputs_O_141;
	::OutputVariables[4,142]	AT %QB."KUKA5_KRC4_ProfiNet_5_0".Module001_8_digital_outputs_O_142;
	::OutputVariables[4,143]	AT %QB."KUKA5_KRC4_ProfiNet_5_0".Module001_8_digital_outputs_O_143;
	::OutputVariables[4,144]	AT %QB."KUKA5_KRC4_ProfiNet_5_0".Module001_8_digital_outputs_O_144;
	::OutputVariables[4,145]	AT %QB."KUKA5_KRC4_ProfiNet_5_0".Module001_8_digital_outputs_O_145;
	::OutputVariables[4,146]	AT %QB."KUKA5_KRC4_ProfiNet_5_0".Module001_8_digital_outputs_O_146;
	::OutputVariables[4,147]	AT %QB."KUKA5_KRC4_ProfiNet_5_0".Module001_8_digital_outputs_O_147;
	::OutputVariables[4,148]	AT %QB."KUKA5_KRC4_ProfiNet_5_0".Module001_8_digital_outputs_O_148;
	::OutputVariables[4,149]	AT %QB."KUKA5_KRC4_ProfiNet_5_0".Module001_8_digital_outputs_O_149;
	::OutputVariables[4,150]	AT %QB."KUKA5_KRC4_ProfiNet_5_0".Module001_8_digital_outputs_O_150;
	::OutputVariables[4,151]	AT %QB."KUKA5_KRC4_ProfiNet_5_0".Module001_8_digital_outputs_O_151;
	::OutputVariables[4,152]	AT %QB."KUKA5_KRC4_ProfiNet_5_0".Module001_8_digital_outputs_O_152;
	::OutputVariables[4,153]	AT %QB."KUKA5_KRC4_ProfiNet_5_0".Module001_8_digital_outputs_O_153;
	::OutputVariables[4,154]	AT %QB."KUKA5_KRC4_ProfiNet_5_0".Module001_8_digital_outputs_O_154;
	::OutputVariables[4,155]	AT %QB."KUKA5_KRC4_ProfiNet_5_0".Module001_8_digital_outputs_O_155;
	::OutputVariables[4,156]	AT %QB."KUKA5_KRC4_ProfiNet_5_0".Module001_8_digital_outputs_O_156;
	::OutputVariables[4,157]	AT %QB."KUKA5_KRC4_ProfiNet_5_0".Module001_8_digital_outputs_O_157;
	::OutputVariables[4,158]	AT %QB."KUKA5_KRC4_ProfiNet_5_0".Module001_8_digital_outputs_O_158;
	::OutputVariables[4,159]	AT %QB."KUKA5_KRC4_ProfiNet_5_0".Module001_8_digital_outputs_O_159;
	::OutputVariables[4,160]	AT %QB."KUKA5_KRC4_ProfiNet_5_0".Module001_8_digital_outputs_O_160;
	::OutputVariables[4,161]	AT %QB."KUKA5_KRC4_ProfiNet_5_0".Module001_8_digital_outputs_O_161;
	::OutputVariables[4,162]	AT %QB."KUKA5_KRC4_ProfiNet_5_0".Module001_8_digital_outputs_O_162;
	::OutputVariables[4,163]	AT %QB."KUKA5_KRC4_ProfiNet_5_0".Module001_8_digital_outputs_O_163;
	::OutputVariables[4,164]	AT %QB."KUKA5_KRC4_ProfiNet_5_0".Module001_8_digital_outputs_O_164;
	::OutputVariables[4,165]	AT %QB."KUKA5_KRC4_ProfiNet_5_0".Module001_8_digital_outputs_O_165;
	::OutputVariables[4,166]	AT %QB."KUKA5_KRC4_ProfiNet_5_0".Module001_8_digital_outputs_O_166;
	::OutputVariables[4,167]	AT %QB."KUKA5_KRC4_ProfiNet_5_0".Module001_8_digital_outputs_O_167;
	::OutputVariables[4,168]	AT %QB."KUKA5_KRC4_ProfiNet_5_0".Module001_8_digital_outputs_O_168;
	::OutputVariables[4,169]	AT %QB."KUKA5_KRC4_ProfiNet_5_0".Module001_8_digital_outputs_O_169;
	::OutputVariables[4,170]	AT %QB."KUKA5_KRC4_ProfiNet_5_0".Module001_8_digital_outputs_O_170;
	::OutputVariables[4,171]	AT %QB."KUKA5_KRC4_ProfiNet_5_0".Module001_8_digital_outputs_O_171;
	::OutputVariables[4,172]	AT %QB."KUKA5_KRC4_ProfiNet_5_0".Module001_8_digital_outputs_O_172;
	::OutputVariables[4,173]	AT %QB."KUKA5_KRC4_ProfiNet_5_0".Module001_8_digital_outputs_O_173;
	::OutputVariables[4,174]	AT %QB."KUKA5_KRC4_ProfiNet_5_0".Module001_8_digital_outputs_O_174;
	::OutputVariables[4,175]	AT %QB."KUKA5_KRC4_ProfiNet_5_0".Module001_8_digital_outputs_O_175;
	::OutputVariables[4,176]	AT %QB."KUKA5_KRC4_ProfiNet_5_0".Module001_8_digital_outputs_O_176;
	::OutputVariables[4,177]	AT %QB."KUKA5_KRC4_ProfiNet_5_0".Module001_8_digital_outputs_O_177;
	::OutputVariables[4,178]	AT %QB."KUKA5_KRC4_ProfiNet_5_0".Module001_8_digital_outputs_O_178;
	::OutputVariables[4,179]	AT %QB."KUKA5_KRC4_ProfiNet_5_0".Module001_8_digital_outputs_O_179;
	::OutputVariables[4,180]	AT %QB."KUKA5_KRC4_ProfiNet_5_0".Module001_8_digital_outputs_O_180;
	::OutputVariables[4,181]	AT %QB."KUKA5_KRC4_ProfiNet_5_0".Module001_8_digital_outputs_O_181;
	::OutputVariables[4,182]	AT %QB."KUKA5_KRC4_ProfiNet_5_0".Module001_8_digital_outputs_O_182;
	::OutputVariables[4,183]	AT %QB."KUKA5_KRC4_ProfiNet_5_0".Module001_8_digital_outputs_O_183;
	::OutputVariables[4,184]	AT %QB."KUKA5_KRC4_ProfiNet_5_0".Module001_8_digital_outputs_O_184;
	::OutputVariables[4,185]	AT %QB."KUKA5_KRC4_ProfiNet_5_0".Module001_8_digital_outputs_O_185;
	::OutputVariables[4,186]	AT %QB."KUKA5_KRC4_ProfiNet_5_0".Module001_8_digital_outputs_O_186;
	::OutputVariables[4,187]	AT %QB."KUKA5_KRC4_ProfiNet_5_0".Module001_8_digital_outputs_O_187;
	::OutputVariables[4,188]	AT %QB."KUKA5_KRC4_ProfiNet_5_0".Module001_8_digital_outputs_O_188;
	::OutputVariables[4,189]	AT %QB."KUKA5_KRC4_ProfiNet_5_0".Module001_8_digital_outputs_O_189;
	::OutputVariables[4,190]	AT %QB."KUKA5_KRC4_ProfiNet_5_0".Module001_8_digital_outputs_O_190;
	::OutputVariables[4,191]	AT %QB."KUKA5_KRC4_ProfiNet_5_0".Module001_8_digital_outputs_O_191;
	::OutputVariables[4,192]	AT %QB."KUKA5_KRC4_ProfiNet_5_0".Module001_8_digital_outputs_O_192;
	::OutputVariables[4,193]	AT %QB."KUKA5_KRC4_ProfiNet_5_0".Module001_8_digital_outputs_O_193;
	::OutputVariables[4,194]	AT %QB."KUKA5_KRC4_ProfiNet_5_0".Module001_8_digital_outputs_O_194;
	::OutputVariables[4,195]	AT %QB."KUKA5_KRC4_ProfiNet_5_0".Module001_8_digital_outputs_O_195;
	::OutputVariables[4,196]	AT %QB."KUKA5_KRC4_ProfiNet_5_0".Module001_8_digital_outputs_O_196;
	::OutputVariables[4,197]	AT %QB."KUKA5_KRC4_ProfiNet_5_0".Module001_8_digital_outputs_O_197;
	::OutputVariables[4,198]	AT %QB."KUKA5_KRC4_ProfiNet_5_0".Module001_8_digital_outputs_O_198;
	::OutputVariables[4,199]	AT %QB."KUKA5_KRC4_ProfiNet_5_0".Module001_8_digital_outputs_O_199;
	::OutputVariables[4,200]	AT %QB."KUKA5_KRC4_ProfiNet_5_0".Module001_8_digital_outputs_O_200;
	::OutputVariables[4,201]	AT %QB."KUKA5_KRC4_ProfiNet_5_0".Module001_8_digital_outputs_O_201;
	::OutputVariables[4,202]	AT %QB."KUKA5_KRC4_ProfiNet_5_0".Module001_8_digital_outputs_O_202;
	::OutputVariables[4,203]	AT %QB."KUKA5_KRC4_ProfiNet_5_0".Module001_8_digital_outputs_O_203;
	::OutputVariables[4,204]	AT %QB."KUKA5_KRC4_ProfiNet_5_0".Module001_8_digital_outputs_O_204;
	::OutputVariables[4,205]	AT %QB."KUKA5_KRC4_ProfiNet_5_0".Module001_8_digital_outputs_O_205;
	::OutputVariables[4,206]	AT %QB."KUKA5_KRC4_ProfiNet_5_0".Module001_8_digital_outputs_O_206;
	::OutputVariables[4,207]	AT %QB."KUKA5_KRC4_ProfiNet_5_0".Module001_8_digital_outputs_O_207;
	::OutputVariables[4,208]	AT %QB."KUKA5_KRC4_ProfiNet_5_0".Module001_8_digital_outputs_O_208;
	::OutputVariables[4,209]	AT %QB."KUKA5_KRC4_ProfiNet_5_0".Module001_8_digital_outputs_O_209;
	::OutputVariables[4,210]	AT %QB."KUKA5_KRC4_ProfiNet_5_0".Module001_8_digital_outputs_O_210;
	::OutputVariables[4,211]	AT %QB."KUKA5_KRC4_ProfiNet_5_0".Module001_8_digital_outputs_O_211;
	::OutputVariables[4,212]	AT %QB."KUKA5_KRC4_ProfiNet_5_0".Module001_8_digital_outputs_O_212;
	::OutputVariables[4,213]	AT %QB."KUKA5_KRC4_ProfiNet_5_0".Module001_8_digital_outputs_O_213;
	::OutputVariables[4,214]	AT %QB."KUKA5_KRC4_ProfiNet_5_0".Module001_8_digital_outputs_O_214;
	::OutputVariables[4,215]	AT %QB."KUKA5_KRC4_ProfiNet_5_0".Module001_8_digital_outputs_O_215;
	::OutputVariables[4,216]	AT %QB."KUKA5_KRC4_ProfiNet_5_0".Module001_8_digital_outputs_O_216;
	::OutputVariables[4,217]	AT %QB."KUKA5_KRC4_ProfiNet_5_0".Module001_8_digital_outputs_O_217;
	::OutputVariables[4,218]	AT %QB."KUKA5_KRC4_ProfiNet_5_0".Module001_8_digital_outputs_O_218;
	::OutputVariables[4,219]	AT %QB."KUKA5_KRC4_ProfiNet_5_0".Module001_8_digital_outputs_O_219;
	::OutputVariables[4,220]	AT %QB."KUKA5_KRC4_ProfiNet_5_0".Module001_8_digital_outputs_O_220;
	::OutputVariables[4,221]	AT %QB."KUKA5_KRC4_ProfiNet_5_0".Module001_8_digital_outputs_O_221;
	::OutputVariables[4,222]	AT %QB."KUKA5_KRC4_ProfiNet_5_0".Module001_8_digital_outputs_O_222;
	::OutputVariables[4,223]	AT %QB."KUKA5_KRC4_ProfiNet_5_0".Module001_8_digital_outputs_O_223;
	::OutputVariables[4,224]	AT %QB."KUKA5_KRC4_ProfiNet_5_0".Module001_8_digital_outputs_O_224;
	::OutputVariables[4,225]	AT %QB."KUKA5_KRC4_ProfiNet_5_0".Module001_8_digital_outputs_O_225;
	::OutputVariables[4,226]	AT %QB."KUKA5_KRC4_ProfiNet_5_0".Module001_8_digital_outputs_O_226;
	::OutputVariables[4,227]	AT %QB."KUKA5_KRC4_ProfiNet_5_0".Module001_8_digital_outputs_O_227;
	::OutputVariables[4,228]	AT %QB."KUKA5_KRC4_ProfiNet_5_0".Module001_8_digital_outputs_O_228;
	::OutputVariables[4,229]	AT %QB."KUKA5_KRC4_ProfiNet_5_0".Module001_8_digital_outputs_O_229;
	::OutputVariables[4,230]	AT %QB."KUKA5_KRC4_ProfiNet_5_0".Module001_8_digital_outputs_O_230;
	::OutputVariables[4,231]	AT %QB."KUKA5_KRC4_ProfiNet_5_0".Module001_8_digital_outputs_O_231;
	::OutputVariables[4,232]	AT %QB."KUKA5_KRC4_ProfiNet_5_0".Module001_8_digital_outputs_O_232;
	::OutputVariables[4,233]	AT %QB."KUKA5_KRC4_ProfiNet_5_0".Module001_8_digital_outputs_O_233;
	::OutputVariables[4,234]	AT %QB."KUKA5_KRC4_ProfiNet_5_0".Module001_8_digital_outputs_O_234;
	::OutputVariables[4,235]	AT %QB."KUKA5_KRC4_ProfiNet_5_0".Module001_8_digital_outputs_O_235;
	::OutputVariables[4,236]	AT %QB."KUKA5_KRC4_ProfiNet_5_0".Module001_8_digital_outputs_O_236;
	::OutputVariables[4,237]	AT %QB."KUKA5_KRC4_ProfiNet_5_0".Module001_8_digital_outputs_O_237;
	::OutputVariables[4,238]	AT %QB."KUKA5_KRC4_ProfiNet_5_0".Module001_8_digital_outputs_O_238;
	::OutputVariables[4,239]	AT %QB."KUKA5_KRC4_ProfiNet_5_0".Module001_8_digital_outputs_O_239;
	::OutputVariables[4,240]	AT %QB."KUKA5_KRC4_ProfiNet_5_0".Module001_8_digital_outputs_O_240;
	::OutputVariables[4,241]	AT %QB."KUKA5_KRC4_ProfiNet_5_0".Module001_8_digital_outputs_O_241;
	::OutputVariables[4,242]	AT %QB."KUKA5_KRC4_ProfiNet_5_0".Module001_8_digital_outputs_O_242;
	::OutputVariables[4,243]	AT %QB."KUKA5_KRC4_ProfiNet_5_0".Module001_8_digital_outputs_O_243;
	::OutputVariables[4,244]	AT %QB."KUKA5_KRC4_ProfiNet_5_0".Module001_8_digital_outputs_O_244;
	::OutputVariables[4,245]	AT %QB."KUKA5_KRC4_ProfiNet_5_0".Module001_8_digital_outputs_O_245;
	::OutputVariables[4,246]	AT %QB."KUKA5_KRC4_ProfiNet_5_0".Module001_8_digital_outputs_O_246;
	::OutputVariables[4,247]	AT %QB."KUKA5_KRC4_ProfiNet_5_0".Module001_8_digital_outputs_O_247;
	::OutputVariables[4,248]	AT %QB."KUKA5_KRC4_ProfiNet_5_0".Module001_8_digital_outputs_O_248;
	::OutputVariables[4,249]	AT %QB."KUKA5_KRC4_ProfiNet_5_0".Module001_8_digital_outputs_O_249;
	::OutputVariables[4,250]	AT %QB."KUKA5_KRC4_ProfiNet_5_0".Module001_8_digital_outputs_O_250;
	::OutputVariables[4,251]	AT %QB."KUKA5_KRC4_ProfiNet_5_0".Module001_8_digital_outputs_O_251;
	::OutputVariables[4,252]	AT %QB."KUKA5_KRC4_ProfiNet_5_0".Module001_8_digital_outputs_O_252;
	::OutputVariables[4,253]	AT %QB."KUKA5_KRC4_ProfiNet_5_0".Module001_8_digital_outputs_O_253;

	(*________________________________________*)
	(*_____________KUKA6 Mappings_____________*)
	(*________________________________________*)

	(*________________________________________*)
	(*_____________KUKA6 Mappings_____________*)
	(*________________________________________*)

	::InputVariables[5,0] AT %IB."KUKA6_KRC5_ProfiNet_6_0".Module001_8_digital_inputs_I_00;
	::InputVariables[5,1] AT %IB."KUKA6_KRC5_ProfiNet_6_0".Module001_8_digital_inputs_I_01;
	::InputVariables[5,2] AT %IB."KUKA6_KRC5_ProfiNet_6_0".Module001_8_digital_inputs_I_02;
	::InputVariables[5,3] AT %IB."KUKA6_KRC5_ProfiNet_6_0".Module001_8_digital_inputs_I_03;
	::InputVariables[5,4] AT %IB."KUKA6_KRC5_ProfiNet_6_0".Module001_8_digital_inputs_I_04;
	::InputVariables[5,5] AT %IB."KUKA6_KRC5_ProfiNet_6_0".Module001_8_digital_inputs_I_05;
	::InputVariables[5,6] AT %IB."KUKA6_KRC5_ProfiNet_6_0".Module001_8_digital_inputs_I_06;
	::InputVariables[5,7] AT %IB."KUKA6_KRC5_ProfiNet_6_0".Module001_8_digital_inputs_I_07;
	::InputVariables[5,8] AT %IB."KUKA6_KRC5_ProfiNet_6_0".Module001_8_digital_inputs_I_08;
	::InputVariables[5,9] AT %IB."KUKA6_KRC5_ProfiNet_6_0".Module001_8_digital_inputs_I_09;
	::InputVariables[5,10] AT %IB."KUKA6_KRC5_ProfiNet_6_0".Module001_8_digital_inputs_I_10;
	::InputVariables[5,11] AT %IB."KUKA6_KRC5_ProfiNet_6_0".Module001_8_digital_inputs_I_11;
	::InputVariables[5,12] AT %IB."KUKA6_KRC5_ProfiNet_6_0".Module001_8_digital_inputs_I_12;
	::InputVariables[5,13] AT %IB."KUKA6_KRC5_ProfiNet_6_0".Module001_8_digital_inputs_I_13;
	::InputVariables[5,14] AT %IB."KUKA6_KRC5_ProfiNet_6_0".Module001_8_digital_inputs_I_14;
	::InputVariables[5,15] AT %IB."KUKA6_KRC5_ProfiNet_6_0".Module001_8_digital_inputs_I_15;
	::InputVariables[5,16] AT %IB."KUKA6_KRC5_ProfiNet_6_0".Module001_8_digital_inputs_I_16;
	::InputVariables[5,17] AT %IB."KUKA6_KRC5_ProfiNet_6_0".Module001_8_digital_inputs_I_17;
	::InputVariables[5,18] AT %IB."KUKA6_KRC5_ProfiNet_6_0".Module001_8_digital_inputs_I_18;
	::InputVariables[5,19] AT %IB."KUKA6_KRC5_ProfiNet_6_0".Module001_8_digital_inputs_I_19;
	::InputVariables[5,20] AT %IB."KUKA6_KRC5_ProfiNet_6_0".Module001_8_digital_inputs_I_20;
	::InputVariables[5,21] AT %IB."KUKA6_KRC5_ProfiNet_6_0".Module001_8_digital_inputs_I_21;
	::InputVariables[5,22] AT %IB."KUKA6_KRC5_ProfiNet_6_0".Module001_8_digital_inputs_I_22;
	::InputVariables[5,23] AT %IB."KUKA6_KRC5_ProfiNet_6_0".Module001_8_digital_inputs_I_23;
	::InputVariables[5,24] AT %IB."KUKA6_KRC5_ProfiNet_6_0".Module001_8_digital_inputs_I_24;
	::InputVariables[5,25] AT %IB."KUKA6_KRC5_ProfiNet_6_0".Module001_8_digital_inputs_I_25;
	::InputVariables[5,26] AT %IB."KUKA6_KRC5_ProfiNet_6_0".Module001_8_digital_inputs_I_26;
	::InputVariables[5,27] AT %IB."KUKA6_KRC5_ProfiNet_6_0".Module001_8_digital_inputs_I_27;
	::InputVariables[5,28] AT %IB."KUKA6_KRC5_ProfiNet_6_0".Module001_8_digital_inputs_I_28;
	::InputVariables[5,29] AT %IB."KUKA6_KRC5_ProfiNet_6_0".Module001_8_digital_inputs_I_29;
	::InputVariables[5,30] AT %IB."KUKA6_KRC5_ProfiNet_6_0".Module001_8_digital_inputs_I_30;
	::InputVariables[5,31] AT %IB."KUKA6_KRC5_ProfiNet_6_0".Module001_8_digital_inputs_I_31;
	::InputVariables[5,32] AT %IB."KUKA6_KRC5_ProfiNet_6_0".Module001_8_digital_inputs_I_32;
	::InputVariables[5,33] AT %IB."KUKA6_KRC5_ProfiNet_6_0".Module001_8_digital_inputs_I_33;
	::InputVariables[5,34] AT %IB."KUKA6_KRC5_ProfiNet_6_0".Module001_8_digital_inputs_I_34;
	::InputVariables[5,35] AT %IB."KUKA6_KRC5_ProfiNet_6_0".Module001_8_digital_inputs_I_35;
	::InputVariables[5,36] AT %IB."KUKA6_KRC5_ProfiNet_6_0".Module001_8_digital_inputs_I_36;
	::InputVariables[5,37] AT %IB."KUKA6_KRC5_ProfiNet_6_0".Module001_8_digital_inputs_I_37;
	::InputVariables[5,38] AT %IB."KUKA6_KRC5_ProfiNet_6_0".Module001_8_digital_inputs_I_38;
	::InputVariables[5,39] AT %IB."KUKA6_KRC5_ProfiNet_6_0".Module001_8_digital_inputs_I_39;
	::InputVariables[5,40] AT %IB."KUKA6_KRC5_ProfiNet_6_0".Module001_8_digital_inputs_I_40;
	::InputVariables[5,41] AT %IB."KUKA6_KRC5_ProfiNet_6_0".Module001_8_digital_inputs_I_41;
	::InputVariables[5,42] AT %IB."KUKA6_KRC5_ProfiNet_6_0".Module001_8_digital_inputs_I_42;
	::InputVariables[5,43] AT %IB."KUKA6_KRC5_ProfiNet_6_0".Module001_8_digital_inputs_I_43;
	::InputVariables[5,44] AT %IB."KUKA6_KRC5_ProfiNet_6_0".Module001_8_digital_inputs_I_44;
	::InputVariables[5,45] AT %IB."KUKA6_KRC5_ProfiNet_6_0".Module001_8_digital_inputs_I_45;
	::InputVariables[5,46] AT %IB."KUKA6_KRC5_ProfiNet_6_0".Module001_8_digital_inputs_I_46;
	::InputVariables[5,47] AT %IB."KUKA6_KRC5_ProfiNet_6_0".Module001_8_digital_inputs_I_47;
	::InputVariables[5,48] AT %IB."KUKA6_KRC5_ProfiNet_6_0".Module001_8_digital_inputs_I_48;
	::InputVariables[5,49] AT %IB."KUKA6_KRC5_ProfiNet_6_0".Module001_8_digital_inputs_I_49;
	::InputVariables[5,50] AT %IB."KUKA6_KRC5_ProfiNet_6_0".Module001_8_digital_inputs_I_50;
	::InputVariables[5,51] AT %IB."KUKA6_KRC5_ProfiNet_6_0".Module001_8_digital_inputs_I_51;
	::InputVariables[5,52] AT %IB."KUKA6_KRC5_ProfiNet_6_0".Module001_8_digital_inputs_I_52;
	::InputVariables[5,53] AT %IB."KUKA6_KRC5_ProfiNet_6_0".Module001_8_digital_inputs_I_53;
	::InputVariables[5,54] AT %IB."KUKA6_KRC5_ProfiNet_6_0".Module001_8_digital_inputs_I_54;
	::InputVariables[5,55] AT %IB."KUKA6_KRC5_ProfiNet_6_0".Module001_8_digital_inputs_I_55;
	::InputVariables[5,56] AT %IB."KUKA6_KRC5_ProfiNet_6_0".Module001_8_digital_inputs_I_56;
	::InputVariables[5,57] AT %IB."KUKA6_KRC5_ProfiNet_6_0".Module001_8_digital_inputs_I_57;
	::InputVariables[5,58] AT %IB."KUKA6_KRC5_ProfiNet_6_0".Module001_8_digital_inputs_I_58;
	::InputVariables[5,59] AT %IB."KUKA6_KRC5_ProfiNet_6_0".Module001_8_digital_inputs_I_59;
	::InputVariables[5,60] AT %IB."KUKA6_KRC5_ProfiNet_6_0".Module001_8_digital_inputs_I_60;
	::InputVariables[5,61] AT %IB."KUKA6_KRC5_ProfiNet_6_0".Module001_8_digital_inputs_I_61;
	::InputVariables[5,62] AT %IB."KUKA6_KRC5_ProfiNet_6_0".Module001_8_digital_inputs_I_62;
	::InputVariables[5,63] AT %IB."KUKA6_KRC5_ProfiNet_6_0".Module001_8_digital_inputs_I_63;
	::InputVariables[5,64] AT %IB."KUKA6_KRC5_ProfiNet_6_0".Module001_8_digital_inputs_I_64;
	::InputVariables[5,65] AT %IB."KUKA6_KRC5_ProfiNet_6_0".Module001_8_digital_inputs_I_65;
	::InputVariables[5,66] AT %IB."KUKA6_KRC5_ProfiNet_6_0".Module001_8_digital_inputs_I_66;
	::InputVariables[5,67] AT %IB."KUKA6_KRC5_ProfiNet_6_0".Module001_8_digital_inputs_I_67;
	::InputVariables[5,68] AT %IB."KUKA6_KRC5_ProfiNet_6_0".Module001_8_digital_inputs_I_68;
	::InputVariables[5,69] AT %IB."KUKA6_KRC5_ProfiNet_6_0".Module001_8_digital_inputs_I_69;
	::InputVariables[5,70] AT %IB."KUKA6_KRC5_ProfiNet_6_0".Module001_8_digital_inputs_I_70;
	::InputVariables[5,71] AT %IB."KUKA6_KRC5_ProfiNet_6_0".Module001_8_digital_inputs_I_71;
	::InputVariables[5,72] AT %IB."KUKA6_KRC5_ProfiNet_6_0".Module001_8_digital_inputs_I_72;
	::InputVariables[5,73] AT %IB."KUKA6_KRC5_ProfiNet_6_0".Module001_8_digital_inputs_I_73;
	::InputVariables[5,74] AT %IB."KUKA6_KRC5_ProfiNet_6_0".Module001_8_digital_inputs_I_74;
	::InputVariables[5,75] AT %IB."KUKA6_KRC5_ProfiNet_6_0".Module001_8_digital_inputs_I_75;
	::InputVariables[5,76] AT %IB."KUKA6_KRC5_ProfiNet_6_0".Module001_8_digital_inputs_I_76;
	::InputVariables[5,77] AT %IB."KUKA6_KRC5_ProfiNet_6_0".Module001_8_digital_inputs_I_77;
	::InputVariables[5,78] AT %IB."KUKA6_KRC5_ProfiNet_6_0".Module001_8_digital_inputs_I_78;
	::InputVariables[5,79] AT %IB."KUKA6_KRC5_ProfiNet_6_0".Module001_8_digital_inputs_I_79;
	::InputVariables[5,80] AT %IB."KUKA6_KRC5_ProfiNet_6_0".Module001_8_digital_inputs_I_80;
	::InputVariables[5,81] AT %IB."KUKA6_KRC5_ProfiNet_6_0".Module001_8_digital_inputs_I_81;
	::InputVariables[5,82] AT %IB."KUKA6_KRC5_ProfiNet_6_0".Module001_8_digital_inputs_I_82;
	::InputVariables[5,83] AT %IB."KUKA6_KRC5_ProfiNet_6_0".Module001_8_digital_inputs_I_83;
	::InputVariables[5,84] AT %IB."KUKA6_KRC5_ProfiNet_6_0".Module001_8_digital_inputs_I_84;
	::InputVariables[5,85] AT %IB."KUKA6_KRC5_ProfiNet_6_0".Module001_8_digital_inputs_I_85;
	::InputVariables[5,86] AT %IB."KUKA6_KRC5_ProfiNet_6_0".Module001_8_digital_inputs_I_86;
	::InputVariables[5,87] AT %IB."KUKA6_KRC5_ProfiNet_6_0".Module001_8_digital_inputs_I_87;
	::InputVariables[5,88] AT %IB."KUKA6_KRC5_ProfiNet_6_0".Module001_8_digital_inputs_I_88;
	::InputVariables[5,89] AT %IB."KUKA6_KRC5_ProfiNet_6_0".Module001_8_digital_inputs_I_89;
	::InputVariables[5,90] AT %IB."KUKA6_KRC5_ProfiNet_6_0".Module001_8_digital_inputs_I_90;
	::InputVariables[5,91] AT %IB."KUKA6_KRC5_ProfiNet_6_0".Module001_8_digital_inputs_I_91;
	::InputVariables[5,92] AT %IB."KUKA6_KRC5_ProfiNet_6_0".Module001_8_digital_inputs_I_92;
	::InputVariables[5,93] AT %IB."KUKA6_KRC5_ProfiNet_6_0".Module001_8_digital_inputs_I_93;
	::InputVariables[5,94] AT %IB."KUKA6_KRC5_ProfiNet_6_0".Module001_8_digital_inputs_I_94;
	::InputVariables[5,95] AT %IB."KUKA6_KRC5_ProfiNet_6_0".Module001_8_digital_inputs_I_95;
	::InputVariables[5,96] AT %IB."KUKA6_KRC5_ProfiNet_6_0".Module001_8_digital_inputs_I_96;
	::InputVariables[5,97] AT %IB."KUKA6_KRC5_ProfiNet_6_0".Module001_8_digital_inputs_I_97;
	::InputVariables[5,98] AT %IB."KUKA6_KRC5_ProfiNet_6_0".Module001_8_digital_inputs_I_98;
	::InputVariables[5,99] AT %IB."KUKA6_KRC5_ProfiNet_6_0".Module001_8_digital_inputs_I_99;
	::InputVariables[5,100] AT %IB."KUKA6_KRC5_ProfiNet_6_0".Module001_8_digital_inputs_I_100;
	::InputVariables[5,101] AT %IB."KUKA6_KRC5_ProfiNet_6_0".Module001_8_digital_inputs_I_101;
	::InputVariables[5,102] AT %IB."KUKA6_KRC5_ProfiNet_6_0".Module001_8_digital_inputs_I_102;
	::InputVariables[5,103] AT %IB."KUKA6_KRC5_ProfiNet_6_0".Module001_8_digital_inputs_I_103;
	::InputVariables[5,104] AT %IB."KUKA6_KRC5_ProfiNet_6_0".Module001_8_digital_inputs_I_104;
	::InputVariables[5,105] AT %IB."KUKA6_KRC5_ProfiNet_6_0".Module001_8_digital_inputs_I_105;
	::InputVariables[5,106] AT %IB."KUKA6_KRC5_ProfiNet_6_0".Module001_8_digital_inputs_I_106;
	::InputVariables[5,107] AT %IB."KUKA6_KRC5_ProfiNet_6_0".Module001_8_digital_inputs_I_107;
	::InputVariables[5,108] AT %IB."KUKA6_KRC5_ProfiNet_6_0".Module001_8_digital_inputs_I_108;
	::InputVariables[5,109] AT %IB."KUKA6_KRC5_ProfiNet_6_0".Module001_8_digital_inputs_I_109;
	::InputVariables[5,110] AT %IB."KUKA6_KRC5_ProfiNet_6_0".Module001_8_digital_inputs_I_110;
	::InputVariables[5,111] AT %IB."KUKA6_KRC5_ProfiNet_6_0".Module001_8_digital_inputs_I_111;
	::InputVariables[5,112] AT %IB."KUKA6_KRC5_ProfiNet_6_0".Module001_8_digital_inputs_I_112;
	::InputVariables[5,113] AT %IB."KUKA6_KRC5_ProfiNet_6_0".Module001_8_digital_inputs_I_113;
	::InputVariables[5,114] AT %IB."KUKA6_KRC5_ProfiNet_6_0".Module001_8_digital_inputs_I_114;
	::InputVariables[5,115] AT %IB."KUKA6_KRC5_ProfiNet_6_0".Module001_8_digital_inputs_I_115;
	::InputVariables[5,116] AT %IB."KUKA6_KRC5_ProfiNet_6_0".Module001_8_digital_inputs_I_116;
	::InputVariables[5,117] AT %IB."KUKA6_KRC5_ProfiNet_6_0".Module001_8_digital_inputs_I_117;
	::InputVariables[5,118] AT %IB."KUKA6_KRC5_ProfiNet_6_0".Module001_8_digital_inputs_I_118;
	::InputVariables[5,119] AT %IB."KUKA6_KRC5_ProfiNet_6_0".Module001_8_digital_inputs_I_119;
	::InputVariables[5,120] AT %IB."KUKA6_KRC5_ProfiNet_6_0".Module001_8_digital_inputs_I_120;
	::InputVariables[5,121] AT %IB."KUKA6_KRC5_ProfiNet_6_0".Module001_8_digital_inputs_I_121;
	::InputVariables[5,122] AT %IB."KUKA6_KRC5_ProfiNet_6_0".Module001_8_digital_inputs_I_122;
	::InputVariables[5,123] AT %IB."KUKA6_KRC5_ProfiNet_6_0".Module001_8_digital_inputs_I_123;
	::InputVariables[5,124] AT %IB."KUKA6_KRC5_ProfiNet_6_0".Module001_8_digital_inputs_I_124;
	::InputVariables[5,125] AT %IB."KUKA6_KRC5_ProfiNet_6_0".Module001_8_digital_inputs_I_125;
	::InputVariables[5,126] AT %IB."KUKA6_KRC5_ProfiNet_6_0".Module001_8_digital_inputs_I_126;
	::InputVariables[5,127] AT %IB."KUKA6_KRC5_ProfiNet_6_0".Module001_8_digital_inputs_I_127;
	::InputVariables[5,128] AT %IB."KUKA6_KRC5_ProfiNet_6_0".Module001_8_digital_inputs_I_128;
	::InputVariables[5,129] AT %IB."KUKA6_KRC5_ProfiNet_6_0".Module001_8_digital_inputs_I_129;
	::InputVariables[5,130] AT %IB."KUKA6_KRC5_ProfiNet_6_0".Module001_8_digital_inputs_I_130;
	::InputVariables[5,131] AT %IB."KUKA6_KRC5_ProfiNet_6_0".Module001_8_digital_inputs_I_131;
	::InputVariables[5,132] AT %IB."KUKA6_KRC5_ProfiNet_6_0".Module001_8_digital_inputs_I_132;
	::InputVariables[5,133] AT %IB."KUKA6_KRC5_ProfiNet_6_0".Module001_8_digital_inputs_I_133;
	::InputVariables[5,134] AT %IB."KUKA6_KRC5_ProfiNet_6_0".Module001_8_digital_inputs_I_134;
	::InputVariables[5,135] AT %IB."KUKA6_KRC5_ProfiNet_6_0".Module001_8_digital_inputs_I_135;
	::InputVariables[5,136] AT %IB."KUKA6_KRC5_ProfiNet_6_0".Module001_8_digital_inputs_I_136;
	::InputVariables[5,137] AT %IB."KUKA6_KRC5_ProfiNet_6_0".Module001_8_digital_inputs_I_137;
	::InputVariables[5,138] AT %IB."KUKA6_KRC5_ProfiNet_6_0".Module001_8_digital_inputs_I_138;
	::InputVariables[5,139] AT %IB."KUKA6_KRC5_ProfiNet_6_0".Module001_8_digital_inputs_I_139;
	::InputVariables[5,140] AT %IB."KUKA6_KRC5_ProfiNet_6_0".Module001_8_digital_inputs_I_140;
	::InputVariables[5,141] AT %IB."KUKA6_KRC5_ProfiNet_6_0".Module001_8_digital_inputs_I_141;
	::InputVariables[5,142] AT %IB."KUKA6_KRC5_ProfiNet_6_0".Module001_8_digital_inputs_I_142;
	::InputVariables[5,143] AT %IB."KUKA6_KRC5_ProfiNet_6_0".Module001_8_digital_inputs_I_143;
	::InputVariables[5,144] AT %IB."KUKA6_KRC5_ProfiNet_6_0".Module001_8_digital_inputs_I_144;
	::InputVariables[5,145] AT %IB."KUKA6_KRC5_ProfiNet_6_0".Module001_8_digital_inputs_I_145;
	::InputVariables[5,146] AT %IB."KUKA6_KRC5_ProfiNet_6_0".Module001_8_digital_inputs_I_146;
	::InputVariables[5,147] AT %IB."KUKA6_KRC5_ProfiNet_6_0".Module001_8_digital_inputs_I_147;
	::InputVariables[5,148] AT %IB."KUKA6_KRC5_ProfiNet_6_0".Module001_8_digital_inputs_I_148;
	::InputVariables[5,149] AT %IB."KUKA6_KRC5_ProfiNet_6_0".Module001_8_digital_inputs_I_149;
	::InputVariables[5,150] AT %IB."KUKA6_KRC5_ProfiNet_6_0".Module001_8_digital_inputs_I_150;
	::InputVariables[5,151] AT %IB."KUKA6_KRC5_ProfiNet_6_0".Module001_8_digital_inputs_I_151;
	::InputVariables[5,152] AT %IB."KUKA6_KRC5_ProfiNet_6_0".Module001_8_digital_inputs_I_152;
	::InputVariables[5,153] AT %IB."KUKA6_KRC5_ProfiNet_6_0".Module001_8_digital_inputs_I_153;
	::InputVariables[5,154] AT %IB."KUKA6_KRC5_ProfiNet_6_0".Module001_8_digital_inputs_I_154;
	::InputVariables[5,155] AT %IB."KUKA6_KRC5_ProfiNet_6_0".Module001_8_digital_inputs_I_155;
	::InputVariables[5,156] AT %IB."KUKA6_KRC5_ProfiNet_6_0".Module001_8_digital_inputs_I_156;
	::InputVariables[5,157] AT %IB."KUKA6_KRC5_ProfiNet_6_0".Module001_8_digital_inputs_I_157;
	::InputVariables[5,158] AT %IB."KUKA6_KRC5_ProfiNet_6_0".Module001_8_digital_inputs_I_158;
	::InputVariables[5,159] AT %IB."KUKA6_KRC5_ProfiNet_6_0".Module001_8_digital_inputs_I_159;
	::InputVariables[5,160] AT %IB."KUKA6_KRC5_ProfiNet_6_0".Module001_8_digital_inputs_I_160;
	::InputVariables[5,161] AT %IB."KUKA6_KRC5_ProfiNet_6_0".Module001_8_digital_inputs_I_161;
	::InputVariables[5,162] AT %IB."KUKA6_KRC5_ProfiNet_6_0".Module001_8_digital_inputs_I_162;
	::InputVariables[5,163] AT %IB."KUKA6_KRC5_ProfiNet_6_0".Module001_8_digital_inputs_I_163;
	::InputVariables[5,164] AT %IB."KUKA6_KRC5_ProfiNet_6_0".Module001_8_digital_inputs_I_164;
	::InputVariables[5,165] AT %IB."KUKA6_KRC5_ProfiNet_6_0".Module001_8_digital_inputs_I_165;
	::InputVariables[5,166] AT %IB."KUKA6_KRC5_ProfiNet_6_0".Module001_8_digital_inputs_I_166;
	::InputVariables[5,167] AT %IB."KUKA6_KRC5_ProfiNet_6_0".Module001_8_digital_inputs_I_167;
	::InputVariables[5,168] AT %IB."KUKA6_KRC5_ProfiNet_6_0".Module001_8_digital_inputs_I_168;
	::InputVariables[5,169] AT %IB."KUKA6_KRC5_ProfiNet_6_0".Module001_8_digital_inputs_I_169;
	::InputVariables[5,170] AT %IB."KUKA6_KRC5_ProfiNet_6_0".Module001_8_digital_inputs_I_170;
	::InputVariables[5,171] AT %IB."KUKA6_KRC5_ProfiNet_6_0".Module001_8_digital_inputs_I_171;
	::InputVariables[5,172] AT %IB."KUKA6_KRC5_ProfiNet_6_0".Module001_8_digital_inputs_I_172;
	::InputVariables[5,173] AT %IB."KUKA6_KRC5_ProfiNet_6_0".Module001_8_digital_inputs_I_173;
	::InputVariables[5,174] AT %IB."KUKA6_KRC5_ProfiNet_6_0".Module001_8_digital_inputs_I_174;
	::InputVariables[5,175] AT %IB."KUKA6_KRC5_ProfiNet_6_0".Module001_8_digital_inputs_I_175;
	::InputVariables[5,176] AT %IB."KUKA6_KRC5_ProfiNet_6_0".Module001_8_digital_inputs_I_176;
	::InputVariables[5,177] AT %IB."KUKA6_KRC5_ProfiNet_6_0".Module001_8_digital_inputs_I_177;
	::InputVariables[5,178] AT %IB."KUKA6_KRC5_ProfiNet_6_0".Module001_8_digital_inputs_I_178;
	::InputVariables[5,179] AT %IB."KUKA6_KRC5_ProfiNet_6_0".Module001_8_digital_inputs_I_179;
	::InputVariables[5,180] AT %IB."KUKA6_KRC5_ProfiNet_6_0".Module001_8_digital_inputs_I_180;
	::InputVariables[5,181] AT %IB."KUKA6_KRC5_ProfiNet_6_0".Module001_8_digital_inputs_I_181;
	::InputVariables[5,182] AT %IB."KUKA6_KRC5_ProfiNet_6_0".Module001_8_digital_inputs_I_182;
	::InputVariables[5,183] AT %IB."KUKA6_KRC5_ProfiNet_6_0".Module001_8_digital_inputs_I_183;
	::InputVariables[5,184] AT %IB."KUKA6_KRC5_ProfiNet_6_0".Module001_8_digital_inputs_I_184;
	::InputVariables[5,185] AT %IB."KUKA6_KRC5_ProfiNet_6_0".Module001_8_digital_inputs_I_185;
	::InputVariables[5,186] AT %IB."KUKA6_KRC5_ProfiNet_6_0".Module001_8_digital_inputs_I_186;
	::InputVariables[5,187] AT %IB."KUKA6_KRC5_ProfiNet_6_0".Module001_8_digital_inputs_I_187;
	::InputVariables[5,188] AT %IB."KUKA6_KRC5_ProfiNet_6_0".Module001_8_digital_inputs_I_188;
	::InputVariables[5,189] AT %IB."KUKA6_KRC5_ProfiNet_6_0".Module001_8_digital_inputs_I_189;
	::InputVariables[5,190] AT %IB."KUKA6_KRC5_ProfiNet_6_0".Module001_8_digital_inputs_I_190;
	::InputVariables[5,191] AT %IB."KUKA6_KRC5_ProfiNet_6_0".Module001_8_digital_inputs_I_191;
	::InputVariables[5,192] AT %IB."KUKA6_KRC5_ProfiNet_6_0".Module001_8_digital_inputs_I_192;
	::InputVariables[5,193] AT %IB."KUKA6_KRC5_ProfiNet_6_0".Module001_8_digital_inputs_I_193;
	::InputVariables[5,194] AT %IB."KUKA6_KRC5_ProfiNet_6_0".Module001_8_digital_inputs_I_194;
	::InputVariables[5,195] AT %IB."KUKA6_KRC5_ProfiNet_6_0".Module001_8_digital_inputs_I_195;
	::InputVariables[5,196] AT %IB."KUKA6_KRC5_ProfiNet_6_0".Module001_8_digital_inputs_I_196;
	::InputVariables[5,197] AT %IB."KUKA6_KRC5_ProfiNet_6_0".Module001_8_digital_inputs_I_197;
	::InputVariables[5,198] AT %IB."KUKA6_KRC5_ProfiNet_6_0".Module001_8_digital_inputs_I_198;
	::InputVariables[5,199] AT %IB."KUKA6_KRC5_ProfiNet_6_0".Module001_8_digital_inputs_I_199;
	::InputVariables[5,200] AT %IB."KUKA6_KRC5_ProfiNet_6_0".Module001_8_digital_inputs_I_200;
	::InputVariables[5,201] AT %IB."KUKA6_KRC5_ProfiNet_6_0".Module001_8_digital_inputs_I_201;
	::InputVariables[5,202] AT %IB."KUKA6_KRC5_ProfiNet_6_0".Module001_8_digital_inputs_I_202;
	::InputVariables[5,203] AT %IB."KUKA6_KRC5_ProfiNet_6_0".Module001_8_digital_inputs_I_203;
	::InputVariables[5,204] AT %IB."KUKA6_KRC5_ProfiNet_6_0".Module001_8_digital_inputs_I_204;
	::InputVariables[5,205] AT %IB."KUKA6_KRC5_ProfiNet_6_0".Module001_8_digital_inputs_I_205;
	::InputVariables[5,206] AT %IB."KUKA6_KRC5_ProfiNet_6_0".Module001_8_digital_inputs_I_206;
	::InputVariables[5,207] AT %IB."KUKA6_KRC5_ProfiNet_6_0".Module001_8_digital_inputs_I_207;
	::InputVariables[5,208] AT %IB."KUKA6_KRC5_ProfiNet_6_0".Module001_8_digital_inputs_I_208;
	::InputVariables[5,209] AT %IB."KUKA6_KRC5_ProfiNet_6_0".Module001_8_digital_inputs_I_209;
	::InputVariables[5,210] AT %IB."KUKA6_KRC5_ProfiNet_6_0".Module001_8_digital_inputs_I_210;
	::InputVariables[5,211] AT %IB."KUKA6_KRC5_ProfiNet_6_0".Module001_8_digital_inputs_I_211;
	::InputVariables[5,212] AT %IB."KUKA6_KRC5_ProfiNet_6_0".Module001_8_digital_inputs_I_212;
	::InputVariables[5,213] AT %IB."KUKA6_KRC5_ProfiNet_6_0".Module001_8_digital_inputs_I_213;
	::InputVariables[5,214] AT %IB."KUKA6_KRC5_ProfiNet_6_0".Module001_8_digital_inputs_I_214;
	::InputVariables[5,215] AT %IB."KUKA6_KRC5_ProfiNet_6_0".Module001_8_digital_inputs_I_215;
	::InputVariables[5,216] AT %IB."KUKA6_KRC5_ProfiNet_6_0".Module001_8_digital_inputs_I_216;
	::InputVariables[5,217] AT %IB."KUKA6_KRC5_ProfiNet_6_0".Module001_8_digital_inputs_I_217;
	::InputVariables[5,218] AT %IB."KUKA6_KRC5_ProfiNet_6_0".Module001_8_digital_inputs_I_218;
	::InputVariables[5,219] AT %IB."KUKA6_KRC5_ProfiNet_6_0".Module001_8_digital_inputs_I_219;
	::InputVariables[5,220] AT %IB."KUKA6_KRC5_ProfiNet_6_0".Module001_8_digital_inputs_I_220;
	::InputVariables[5,221] AT %IB."KUKA6_KRC5_ProfiNet_6_0".Module001_8_digital_inputs_I_221;
	::InputVariables[5,222] AT %IB."KUKA6_KRC5_ProfiNet_6_0".Module001_8_digital_inputs_I_222;
	::InputVariables[5,223] AT %IB."KUKA6_KRC5_ProfiNet_6_0".Module001_8_digital_inputs_I_223;
	::InputVariables[5,224] AT %IB."KUKA6_KRC5_ProfiNet_6_0".Module001_8_digital_inputs_I_224;
	::InputVariables[5,225] AT %IB."KUKA6_KRC5_ProfiNet_6_0".Module001_8_digital_inputs_I_225;
	::InputVariables[5,226] AT %IB."KUKA6_KRC5_ProfiNet_6_0".Module001_8_digital_inputs_I_226;
	::InputVariables[5,227] AT %IB."KUKA6_KRC5_ProfiNet_6_0".Module001_8_digital_inputs_I_227;
	::InputVariables[5,228] AT %IB."KUKA6_KRC5_ProfiNet_6_0".Module001_8_digital_inputs_I_228;
	::InputVariables[5,229] AT %IB."KUKA6_KRC5_ProfiNet_6_0".Module001_8_digital_inputs_I_229;
	::InputVariables[5,230] AT %IB."KUKA6_KRC5_ProfiNet_6_0".Module001_8_digital_inputs_I_230;
	::InputVariables[5,231] AT %IB."KUKA6_KRC5_ProfiNet_6_0".Module001_8_digital_inputs_I_231;
	::InputVariables[5,232] AT %IB."KUKA6_KRC5_ProfiNet_6_0".Module001_8_digital_inputs_I_232;
	::InputVariables[5,233] AT %IB."KUKA6_KRC5_ProfiNet_6_0".Module001_8_digital_inputs_I_233;
	::InputVariables[5,234] AT %IB."KUKA6_KRC5_ProfiNet_6_0".Module001_8_digital_inputs_I_234;
	::InputVariables[5,235] AT %IB."KUKA6_KRC5_ProfiNet_6_0".Module001_8_digital_inputs_I_235;
	::InputVariables[5,236] AT %IB."KUKA6_KRC5_ProfiNet_6_0".Module001_8_digital_inputs_I_236;
	::InputVariables[5,237] AT %IB."KUKA6_KRC5_ProfiNet_6_0".Module001_8_digital_inputs_I_237;
	::InputVariables[5,238] AT %IB."KUKA6_KRC5_ProfiNet_6_0".Module001_8_digital_inputs_I_238;
	::InputVariables[5,239] AT %IB."KUKA6_KRC5_ProfiNet_6_0".Module001_8_digital_inputs_I_239;
	::InputVariables[5,240] AT %IB."KUKA6_KRC5_ProfiNet_6_0".Module001_8_digital_inputs_I_240;
	::InputVariables[5,241] AT %IB."KUKA6_KRC5_ProfiNet_6_0".Module001_8_digital_inputs_I_241;
	::InputVariables[5,242] AT %IB."KUKA6_KRC5_ProfiNet_6_0".Module001_8_digital_inputs_I_242;
	::InputVariables[5,243] AT %IB."KUKA6_KRC5_ProfiNet_6_0".Module001_8_digital_inputs_I_243;
	::InputVariables[5,244] AT %IB."KUKA6_KRC5_ProfiNet_6_0".Module001_8_digital_inputs_I_244;
	::InputVariables[5,245] AT %IB."KUKA6_KRC5_ProfiNet_6_0".Module001_8_digital_inputs_I_245;
	::InputVariables[5,246] AT %IB."KUKA6_KRC5_ProfiNet_6_0".Module001_8_digital_inputs_I_246;
	::InputVariables[5,247] AT %IB."KUKA6_KRC5_ProfiNet_6_0".Module001_8_digital_inputs_I_247;
	::InputVariables[5,248] AT %IB."KUKA6_KRC5_ProfiNet_6_0".Module001_8_digital_inputs_I_248;
	::InputVariables[5,249] AT %IB."KUKA6_KRC5_ProfiNet_6_0".Module001_8_digital_inputs_I_249;
	::InputVariables[5,250] AT %IB."KUKA6_KRC5_ProfiNet_6_0".Module001_8_digital_inputs_I_250;
	::InputVariables[5,251] AT %IB."KUKA6_KRC5_ProfiNet_6_0".Module001_8_digital_inputs_I_251;
	::InputVariables[5,252] AT %IB."KUKA6_KRC5_ProfiNet_6_0".Module001_8_digital_inputs_I_252;
	::InputVariables[5,253] AT %IB."KUKA6_KRC5_ProfiNet_6_0".Module001_8_digital_inputs_I_253;

	::OutputVariables[5,0]	AT %QB."KUKA6_KRC5_ProfiNet_6_0".Module001_8_digital_outputs_O_00;
	::OutputVariables[5,1]	AT %QB."KUKA6_KRC5_ProfiNet_6_0".Module001_8_digital_outputs_O_01;
	::OutputVariables[5,2]	AT %QB."KUKA6_KRC5_ProfiNet_6_0".Module001_8_digital_outputs_O_02;
	::OutputVariables[5,3]	AT %QB."KUKA6_KRC5_ProfiNet_6_0".Module001_8_digital_outputs_O_03;
	::OutputVariables[5,4]	AT %QB."KUKA6_KRC5_ProfiNet_6_0".Module001_8_digital_outputs_O_04;
	::OutputVariables[5,5]	AT %QB."KUKA6_KRC5_ProfiNet_6_0".Module001_8_digital_outputs_O_05;
	::OutputVariables[5,6]	AT %QB."KUKA6_KRC5_ProfiNet_6_0".Module001_8_digital_outputs_O_06;
	::OutputVariables[5,7]	AT %QB."KUKA6_KRC5_ProfiNet_6_0".Module001_8_digital_outputs_O_07;
	::OutputVariables[5,8]	AT %QB."KUKA6_KRC5_ProfiNet_6_0".Module001_8_digital_outputs_O_08;
	::OutputVariables[5,9]	AT %QB."KUKA6_KRC5_ProfiNet_6_0".Module001_8_digital_outputs_O_09;
	::OutputVariables[5,10]	AT %QB."KUKA6_KRC5_ProfiNet_6_0".Module001_8_digital_outputs_O_10;
	::OutputVariables[5,11]	AT %QB."KUKA6_KRC5_ProfiNet_6_0".Module001_8_digital_outputs_O_11;
	::OutputVariables[5,12]	AT %QB."KUKA6_KRC5_ProfiNet_6_0".Module001_8_digital_outputs_O_12;
	::OutputVariables[5,13]	AT %QB."KUKA6_KRC5_ProfiNet_6_0".Module001_8_digital_outputs_O_13;
	::OutputVariables[5,14]	AT %QB."KUKA6_KRC5_ProfiNet_6_0".Module001_8_digital_outputs_O_14;
	::OutputVariables[5,15]	AT %QB."KUKA6_KRC5_ProfiNet_6_0".Module001_8_digital_outputs_O_15;
	::OutputVariables[5,16]	AT %QB."KUKA6_KRC5_ProfiNet_6_0".Module001_8_digital_outputs_O_16;
	::OutputVariables[5,17]	AT %QB."KUKA6_KRC5_ProfiNet_6_0".Module001_8_digital_outputs_O_17;
	::OutputVariables[5,18]	AT %QB."KUKA6_KRC5_ProfiNet_6_0".Module001_8_digital_outputs_O_18;
	::OutputVariables[5,19]	AT %QB."KUKA6_KRC5_ProfiNet_6_0".Module001_8_digital_outputs_O_19;
	::OutputVariables[5,20]	AT %QB."KUKA6_KRC5_ProfiNet_6_0".Module001_8_digital_outputs_O_20;
	::OutputVariables[5,21]	AT %QB."KUKA6_KRC5_ProfiNet_6_0".Module001_8_digital_outputs_O_21;
	::OutputVariables[5,22]	AT %QB."KUKA6_KRC5_ProfiNet_6_0".Module001_8_digital_outputs_O_22;
	::OutputVariables[5,23]	AT %QB."KUKA6_KRC5_ProfiNet_6_0".Module001_8_digital_outputs_O_23;
	::OutputVariables[5,24]	AT %QB."KUKA6_KRC5_ProfiNet_6_0".Module001_8_digital_outputs_O_24;
	::OutputVariables[5,25]	AT %QB."KUKA6_KRC5_ProfiNet_6_0".Module001_8_digital_outputs_O_25;
	::OutputVariables[5,26]	AT %QB."KUKA6_KRC5_ProfiNet_6_0".Module001_8_digital_outputs_O_26;
	::OutputVariables[5,27]	AT %QB."KUKA6_KRC5_ProfiNet_6_0".Module001_8_digital_outputs_O_27;
	::OutputVariables[5,28]	AT %QB."KUKA6_KRC5_ProfiNet_6_0".Module001_8_digital_outputs_O_28;
	::OutputVariables[5,29]	AT %QB."KUKA6_KRC5_ProfiNet_6_0".Module001_8_digital_outputs_O_29;
	::OutputVariables[5,30]	AT %QB."KUKA6_KRC5_ProfiNet_6_0".Module001_8_digital_outputs_O_30;
	::OutputVariables[5,31]	AT %QB."KUKA6_KRC5_ProfiNet_6_0".Module001_8_digital_outputs_O_31;
	::OutputVariables[5,32]	AT %QB."KUKA6_KRC5_ProfiNet_6_0".Module001_8_digital_outputs_O_32;
	::OutputVariables[5,33]	AT %QB."KUKA6_KRC5_ProfiNet_6_0".Module001_8_digital_outputs_O_33;
	::OutputVariables[5,34]	AT %QB."KUKA6_KRC5_ProfiNet_6_0".Module001_8_digital_outputs_O_34;
	::OutputVariables[5,35]	AT %QB."KUKA6_KRC5_ProfiNet_6_0".Module001_8_digital_outputs_O_35;
	::OutputVariables[5,36]	AT %QB."KUKA6_KRC5_ProfiNet_6_0".Module001_8_digital_outputs_O_36;
	::OutputVariables[5,37]	AT %QB."KUKA6_KRC5_ProfiNet_6_0".Module001_8_digital_outputs_O_37;
	::OutputVariables[5,38]	AT %QB."KUKA6_KRC5_ProfiNet_6_0".Module001_8_digital_outputs_O_38;
	::OutputVariables[5,39]	AT %QB."KUKA6_KRC5_ProfiNet_6_0".Module001_8_digital_outputs_O_39;
	::OutputVariables[5,40]	AT %QB."KUKA6_KRC5_ProfiNet_6_0".Module001_8_digital_outputs_O_40;
	::OutputVariables[5,41]	AT %QB."KUKA6_KRC5_ProfiNet_6_0".Module001_8_digital_outputs_O_41;
	::OutputVariables[5,42]	AT %QB."KUKA6_KRC5_ProfiNet_6_0".Module001_8_digital_outputs_O_42;
	::OutputVariables[5,43]	AT %QB."KUKA6_KRC5_ProfiNet_6_0".Module001_8_digital_outputs_O_43;
	::OutputVariables[5,44]	AT %QB."KUKA6_KRC5_ProfiNet_6_0".Module001_8_digital_outputs_O_44;
	::OutputVariables[5,45]	AT %QB."KUKA6_KRC5_ProfiNet_6_0".Module001_8_digital_outputs_O_45;
	::OutputVariables[5,46]	AT %QB."KUKA6_KRC5_ProfiNet_6_0".Module001_8_digital_outputs_O_46;
	::OutputVariables[5,47]	AT %QB."KUKA6_KRC5_ProfiNet_6_0".Module001_8_digital_outputs_O_47;
	::OutputVariables[5,48]	AT %QB."KUKA6_KRC5_ProfiNet_6_0".Module001_8_digital_outputs_O_48;
	::OutputVariables[5,49]	AT %QB."KUKA6_KRC5_ProfiNet_6_0".Module001_8_digital_outputs_O_49;
	::OutputVariables[5,50]	AT %QB."KUKA6_KRC5_ProfiNet_6_0".Module001_8_digital_outputs_O_50;
	::OutputVariables[5,51]	AT %QB."KUKA6_KRC5_ProfiNet_6_0".Module001_8_digital_outputs_O_51;
	::OutputVariables[5,52]	AT %QB."KUKA6_KRC5_ProfiNet_6_0".Module001_8_digital_outputs_O_52;
	::OutputVariables[5,53]	AT %QB."KUKA6_KRC5_ProfiNet_6_0".Module001_8_digital_outputs_O_53;
	::OutputVariables[5,54]	AT %QB."KUKA6_KRC5_ProfiNet_6_0".Module001_8_digital_outputs_O_54;
	::OutputVariables[5,55]	AT %QB."KUKA6_KRC5_ProfiNet_6_0".Module001_8_digital_outputs_O_55;
	::OutputVariables[5,56]	AT %QB."KUKA6_KRC5_ProfiNet_6_0".Module001_8_digital_outputs_O_56;
	::OutputVariables[5,57]	AT %QB."KUKA6_KRC5_ProfiNet_6_0".Module001_8_digital_outputs_O_57;
	::OutputVariables[5,58]	AT %QB."KUKA6_KRC5_ProfiNet_6_0".Module001_8_digital_outputs_O_58;
	::OutputVariables[5,59]	AT %QB."KUKA6_KRC5_ProfiNet_6_0".Module001_8_digital_outputs_O_59;
	::OutputVariables[5,60]	AT %QB."KUKA6_KRC5_ProfiNet_6_0".Module001_8_digital_outputs_O_60;
	::OutputVariables[5,61]	AT %QB."KUKA6_KRC5_ProfiNet_6_0".Module001_8_digital_outputs_O_61;
	::OutputVariables[5,62]	AT %QB."KUKA6_KRC5_ProfiNet_6_0".Module001_8_digital_outputs_O_62;
	::OutputVariables[5,63]	AT %QB."KUKA6_KRC5_ProfiNet_6_0".Module001_8_digital_outputs_O_63;
	::OutputVariables[5,64]	AT %QB."KUKA6_KRC5_ProfiNet_6_0".Module001_8_digital_outputs_O_64;
	::OutputVariables[5,65]	AT %QB."KUKA6_KRC5_ProfiNet_6_0".Module001_8_digital_outputs_O_65;
	::OutputVariables[5,66]	AT %QB."KUKA6_KRC5_ProfiNet_6_0".Module001_8_digital_outputs_O_66;
	::OutputVariables[5,67]	AT %QB."KUKA6_KRC5_ProfiNet_6_0".Module001_8_digital_outputs_O_67;
	::OutputVariables[5,68]	AT %QB."KUKA6_KRC5_ProfiNet_6_0".Module001_8_digital_outputs_O_68;
	::OutputVariables[5,69]	AT %QB."KUKA6_KRC5_ProfiNet_6_0".Module001_8_digital_outputs_O_69;
	::OutputVariables[5,70]	AT %QB."KUKA6_KRC5_ProfiNet_6_0".Module001_8_digital_outputs_O_70;
	::OutputVariables[5,71]	AT %QB."KUKA6_KRC5_ProfiNet_6_0".Module001_8_digital_outputs_O_71;
	::OutputVariables[5,72]	AT %QB."KUKA6_KRC5_ProfiNet_6_0".Module001_8_digital_outputs_O_72;
	::OutputVariables[5,73]	AT %QB."KUKA6_KRC5_ProfiNet_6_0".Module001_8_digital_outputs_O_73;
	::OutputVariables[5,74]	AT %QB."KUKA6_KRC5_ProfiNet_6_0".Module001_8_digital_outputs_O_74;
	::OutputVariables[5,75]	AT %QB."KUKA6_KRC5_ProfiNet_6_0".Module001_8_digital_outputs_O_75;
	::OutputVariables[5,76]	AT %QB."KUKA6_KRC5_ProfiNet_6_0".Module001_8_digital_outputs_O_76;
	::OutputVariables[5,77]	AT %QB."KUKA6_KRC5_ProfiNet_6_0".Module001_8_digital_outputs_O_77;
	::OutputVariables[5,78]	AT %QB."KUKA6_KRC5_ProfiNet_6_0".Module001_8_digital_outputs_O_78;
	::OutputVariables[5,79]	AT %QB."KUKA6_KRC5_ProfiNet_6_0".Module001_8_digital_outputs_O_79;
	::OutputVariables[5,80]	AT %QB."KUKA6_KRC5_ProfiNet_6_0".Module001_8_digital_outputs_O_80;
	::OutputVariables[5,81]	AT %QB."KUKA6_KRC5_ProfiNet_6_0".Module001_8_digital_outputs_O_81;
	::OutputVariables[5,82]	AT %QB."KUKA6_KRC5_ProfiNet_6_0".Module001_8_digital_outputs_O_82;
	::OutputVariables[5,83]	AT %QB."KUKA6_KRC5_ProfiNet_6_0".Module001_8_digital_outputs_O_83;
	::OutputVariables[5,84]	AT %QB."KUKA6_KRC5_ProfiNet_6_0".Module001_8_digital_outputs_O_84;
	::OutputVariables[5,85]	AT %QB."KUKA6_KRC5_ProfiNet_6_0".Module001_8_digital_outputs_O_85;
	::OutputVariables[5,86]	AT %QB."KUKA6_KRC5_ProfiNet_6_0".Module001_8_digital_outputs_O_86;
	::OutputVariables[5,87]	AT %QB."KUKA6_KRC5_ProfiNet_6_0".Module001_8_digital_outputs_O_87;
	::OutputVariables[5,88]	AT %QB."KUKA6_KRC5_ProfiNet_6_0".Module001_8_digital_outputs_O_88;
	::OutputVariables[5,89]	AT %QB."KUKA6_KRC5_ProfiNet_6_0".Module001_8_digital_outputs_O_89;
	::OutputVariables[5,90]	AT %QB."KUKA6_KRC5_ProfiNet_6_0".Module001_8_digital_outputs_O_90;
	::OutputVariables[5,91]	AT %QB."KUKA6_KRC5_ProfiNet_6_0".Module001_8_digital_outputs_O_91;
	::OutputVariables[5,92]	AT %QB."KUKA6_KRC5_ProfiNet_6_0".Module001_8_digital_outputs_O_92;
	::OutputVariables[5,93]	AT %QB."KUKA6_KRC5_ProfiNet_6_0".Module001_8_digital_outputs_O_93;
	::OutputVariables[5,94]	AT %QB."KUKA6_KRC5_ProfiNet_6_0".Module001_8_digital_outputs_O_94;
	::OutputVariables[5,95]	AT %QB."KUKA6_KRC5_ProfiNet_6_0".Module001_8_digital_outputs_O_95;
	::OutputVariables[5,96]	AT %QB."KUKA6_KRC5_ProfiNet_6_0".Module001_8_digital_outputs_O_96;
	::OutputVariables[5,97]	AT %QB."KUKA6_KRC5_ProfiNet_6_0".Module001_8_digital_outputs_O_97;
	::OutputVariables[5,98]	AT %QB."KUKA6_KRC5_ProfiNet_6_0".Module001_8_digital_outputs_O_98;
	::OutputVariables[5,99]	AT %QB."KUKA6_KRC5_ProfiNet_6_0".Module001_8_digital_outputs_O_99;
	::OutputVariables[5,100]	AT %QB."KUKA6_KRC5_ProfiNet_6_0".Module001_8_digital_outputs_O_100;
	::OutputVariables[5,101]	AT %QB."KUKA6_KRC5_ProfiNet_6_0".Module001_8_digital_outputs_O_101;
	::OutputVariables[5,102]	AT %QB."KUKA6_KRC5_ProfiNet_6_0".Module001_8_digital_outputs_O_102;
	::OutputVariables[5,103]	AT %QB."KUKA6_KRC5_ProfiNet_6_0".Module001_8_digital_outputs_O_103;
	::OutputVariables[5,104]	AT %QB."KUKA6_KRC5_ProfiNet_6_0".Module001_8_digital_outputs_O_104;
	::OutputVariables[5,105]	AT %QB."KUKA6_KRC5_ProfiNet_6_0".Module001_8_digital_outputs_O_105;
	::OutputVariables[5,106]	AT %QB."KUKA6_KRC5_ProfiNet_6_0".Module001_8_digital_outputs_O_106;
	::OutputVariables[5,107]	AT %QB."KUKA6_KRC5_ProfiNet_6_0".Module001_8_digital_outputs_O_107;
	::OutputVariables[5,108]	AT %QB."KUKA6_KRC5_ProfiNet_6_0".Module001_8_digital_outputs_O_108;
	::OutputVariables[5,109]	AT %QB."KUKA6_KRC5_ProfiNet_6_0".Module001_8_digital_outputs_O_109;
	::OutputVariables[5,110]	AT %QB."KUKA6_KRC5_ProfiNet_6_0".Module001_8_digital_outputs_O_110;
	::OutputVariables[5,111]	AT %QB."KUKA6_KRC5_ProfiNet_6_0".Module001_8_digital_outputs_O_111;
	::OutputVariables[5,112]	AT %QB."KUKA6_KRC5_ProfiNet_6_0".Module001_8_digital_outputs_O_112;
	::OutputVariables[5,113]	AT %QB."KUKA6_KRC5_ProfiNet_6_0".Module001_8_digital_outputs_O_113;
	::OutputVariables[5,114]	AT %QB."KUKA6_KRC5_ProfiNet_6_0".Module001_8_digital_outputs_O_114;
	::OutputVariables[5,115]	AT %QB."KUKA6_KRC5_ProfiNet_6_0".Module001_8_digital_outputs_O_115;
	::OutputVariables[5,116]	AT %QB."KUKA6_KRC5_ProfiNet_6_0".Module001_8_digital_outputs_O_116;
	::OutputVariables[5,117]	AT %QB."KUKA6_KRC5_ProfiNet_6_0".Module001_8_digital_outputs_O_117;
	::OutputVariables[5,118]	AT %QB."KUKA6_KRC5_ProfiNet_6_0".Module001_8_digital_outputs_O_118;
	::OutputVariables[5,119]	AT %QB."KUKA6_KRC5_ProfiNet_6_0".Module001_8_digital_outputs_O_119;
	::OutputVariables[5,120]	AT %QB."KUKA6_KRC5_ProfiNet_6_0".Module001_8_digital_outputs_O_120;
	::OutputVariables[5,121]	AT %QB."KUKA6_KRC5_ProfiNet_6_0".Module001_8_digital_outputs_O_121;
	::OutputVariables[5,122]	AT %QB."KUKA6_KRC5_ProfiNet_6_0".Module001_8_digital_outputs_O_122;
	::OutputVariables[5,123]	AT %QB."KUKA6_KRC5_ProfiNet_6_0".Module001_8_digital_outputs_O_123;
	::OutputVariables[5,124]	AT %QB."KUKA6_KRC5_ProfiNet_6_0".Module001_8_digital_outputs_O_124;
	::OutputVariables[5,125]	AT %QB."KUKA6_KRC5_ProfiNet_6_0".Module001_8_digital_outputs_O_125;
	::OutputVariables[5,126]	AT %QB."KUKA6_KRC5_ProfiNet_6_0".Module001_8_digital_outputs_O_126;
	::OutputVariables[5,127]	AT %QB."KUKA6_KRC5_ProfiNet_6_0".Module001_8_digital_outputs_O_127;
	::OutputVariables[5,128]	AT %QB."KUKA6_KRC5_ProfiNet_6_0".Module001_8_digital_outputs_O_128;
	::OutputVariables[5,129]	AT %QB."KUKA6_KRC5_ProfiNet_6_0".Module001_8_digital_outputs_O_129;
	::OutputVariables[5,130]	AT %QB."KUKA6_KRC5_ProfiNet_6_0".Module001_8_digital_outputs_O_130;
	::OutputVariables[5,131]	AT %QB."KUKA6_KRC5_ProfiNet_6_0".Module001_8_digital_outputs_O_131;
	::OutputVariables[5,132]	AT %QB."KUKA6_KRC5_ProfiNet_6_0".Module001_8_digital_outputs_O_132;
	::OutputVariables[5,133]	AT %QB."KUKA6_KRC5_ProfiNet_6_0".Module001_8_digital_outputs_O_133;
	::OutputVariables[5,134]	AT %QB."KUKA6_KRC5_ProfiNet_6_0".Module001_8_digital_outputs_O_134;
	::OutputVariables[5,135]	AT %QB."KUKA6_KRC5_ProfiNet_6_0".Module001_8_digital_outputs_O_135;
	::OutputVariables[5,136]	AT %QB."KUKA6_KRC5_ProfiNet_6_0".Module001_8_digital_outputs_O_136;
	::OutputVariables[5,137]	AT %QB."KUKA6_KRC5_ProfiNet_6_0".Module001_8_digital_outputs_O_137;
	::OutputVariables[5,138]	AT %QB."KUKA6_KRC5_ProfiNet_6_0".Module001_8_digital_outputs_O_138;
	::OutputVariables[5,139]	AT %QB."KUKA6_KRC5_ProfiNet_6_0".Module001_8_digital_outputs_O_139;
	::OutputVariables[5,140]	AT %QB."KUKA6_KRC5_ProfiNet_6_0".Module001_8_digital_outputs_O_140;
	::OutputVariables[5,141]	AT %QB."KUKA6_KRC5_ProfiNet_6_0".Module001_8_digital_outputs_O_141;
	::OutputVariables[5,142]	AT %QB."KUKA6_KRC5_ProfiNet_6_0".Module001_8_digital_outputs_O_142;
	::OutputVariables[5,143]	AT %QB."KUKA6_KRC5_ProfiNet_6_0".Module001_8_digital_outputs_O_143;
	::OutputVariables[5,144]	AT %QB."KUKA6_KRC5_ProfiNet_6_0".Module001_8_digital_outputs_O_144;
	::OutputVariables[5,145]	AT %QB."KUKA6_KRC5_ProfiNet_6_0".Module001_8_digital_outputs_O_145;
	::OutputVariables[5,146]	AT %QB."KUKA6_KRC5_ProfiNet_6_0".Module001_8_digital_outputs_O_146;
	::OutputVariables[5,147]	AT %QB."KUKA6_KRC5_ProfiNet_6_0".Module001_8_digital_outputs_O_147;
	::OutputVariables[5,148]	AT %QB."KUKA6_KRC5_ProfiNet_6_0".Module001_8_digital_outputs_O_148;
	::OutputVariables[5,149]	AT %QB."KUKA6_KRC5_ProfiNet_6_0".Module001_8_digital_outputs_O_149;
	::OutputVariables[5,150]	AT %QB."KUKA6_KRC5_ProfiNet_6_0".Module001_8_digital_outputs_O_150;
	::OutputVariables[5,151]	AT %QB."KUKA6_KRC5_ProfiNet_6_0".Module001_8_digital_outputs_O_151;
	::OutputVariables[5,152]	AT %QB."KUKA6_KRC5_ProfiNet_6_0".Module001_8_digital_outputs_O_152;
	::OutputVariables[5,153]	AT %QB."KUKA6_KRC5_ProfiNet_6_0".Module001_8_digital_outputs_O_153;
	::OutputVariables[5,154]	AT %QB."KUKA6_KRC5_ProfiNet_6_0".Module001_8_digital_outputs_O_154;
	::OutputVariables[5,155]	AT %QB."KUKA6_KRC5_ProfiNet_6_0".Module001_8_digital_outputs_O_155;
	::OutputVariables[5,156]	AT %QB."KUKA6_KRC5_ProfiNet_6_0".Module001_8_digital_outputs_O_156;
	::OutputVariables[5,157]	AT %QB."KUKA6_KRC5_ProfiNet_6_0".Module001_8_digital_outputs_O_157;
	::OutputVariables[5,158]	AT %QB."KUKA6_KRC5_ProfiNet_6_0".Module001_8_digital_outputs_O_158;
	::OutputVariables[5,159]	AT %QB."KUKA6_KRC5_ProfiNet_6_0".Module001_8_digital_outputs_O_159;
	::OutputVariables[5,160]	AT %QB."KUKA6_KRC5_ProfiNet_6_0".Module001_8_digital_outputs_O_160;
	::OutputVariables[5,161]	AT %QB."KUKA6_KRC5_ProfiNet_6_0".Module001_8_digital_outputs_O_161;
	::OutputVariables[5,162]	AT %QB."KUKA6_KRC5_ProfiNet_6_0".Module001_8_digital_outputs_O_162;
	::OutputVariables[5,163]	AT %QB."KUKA6_KRC5_ProfiNet_6_0".Module001_8_digital_outputs_O_163;
	::OutputVariables[5,164]	AT %QB."KUKA6_KRC5_ProfiNet_6_0".Module001_8_digital_outputs_O_164;
	::OutputVariables[5,165]	AT %QB."KUKA6_KRC5_ProfiNet_6_0".Module001_8_digital_outputs_O_165;
	::OutputVariables[5,166]	AT %QB."KUKA6_KRC5_ProfiNet_6_0".Module001_8_digital_outputs_O_166;
	::OutputVariables[5,167]	AT %QB."KUKA6_KRC5_ProfiNet_6_0".Module001_8_digital_outputs_O_167;
	::OutputVariables[5,168]	AT %QB."KUKA6_KRC5_ProfiNet_6_0".Module001_8_digital_outputs_O_168;
	::OutputVariables[5,169]	AT %QB."KUKA6_KRC5_ProfiNet_6_0".Module001_8_digital_outputs_O_169;
	::OutputVariables[5,170]	AT %QB."KUKA6_KRC5_ProfiNet_6_0".Module001_8_digital_outputs_O_170;
	::OutputVariables[5,171]	AT %QB."KUKA6_KRC5_ProfiNet_6_0".Module001_8_digital_outputs_O_171;
	::OutputVariables[5,172]	AT %QB."KUKA6_KRC5_ProfiNet_6_0".Module001_8_digital_outputs_O_172;
	::OutputVariables[5,173]	AT %QB."KUKA6_KRC5_ProfiNet_6_0".Module001_8_digital_outputs_O_173;
	::OutputVariables[5,174]	AT %QB."KUKA6_KRC5_ProfiNet_6_0".Module001_8_digital_outputs_O_174;
	::OutputVariables[5,175]	AT %QB."KUKA6_KRC5_ProfiNet_6_0".Module001_8_digital_outputs_O_175;
	::OutputVariables[5,176]	AT %QB."KUKA6_KRC5_ProfiNet_6_0".Module001_8_digital_outputs_O_176;
	::OutputVariables[5,177]	AT %QB."KUKA6_KRC5_ProfiNet_6_0".Module001_8_digital_outputs_O_177;
	::OutputVariables[5,178]	AT %QB."KUKA6_KRC5_ProfiNet_6_0".Module001_8_digital_outputs_O_178;
	::OutputVariables[5,179]	AT %QB."KUKA6_KRC5_ProfiNet_6_0".Module001_8_digital_outputs_O_179;
	::OutputVariables[5,180]	AT %QB."KUKA6_KRC5_ProfiNet_6_0".Module001_8_digital_outputs_O_180;
	::OutputVariables[5,181]	AT %QB."KUKA6_KRC5_ProfiNet_6_0".Module001_8_digital_outputs_O_181;
	::OutputVariables[5,182]	AT %QB."KUKA6_KRC5_ProfiNet_6_0".Module001_8_digital_outputs_O_182;
	::OutputVariables[5,183]	AT %QB."KUKA6_KRC5_ProfiNet_6_0".Module001_8_digital_outputs_O_183;
	::OutputVariables[5,184]	AT %QB."KUKA6_KRC5_ProfiNet_6_0".Module001_8_digital_outputs_O_184;
	::OutputVariables[5,185]	AT %QB."KUKA6_KRC5_ProfiNet_6_0".Module001_8_digital_outputs_O_185;
	::OutputVariables[5,186]	AT %QB."KUKA6_KRC5_ProfiNet_6_0".Module001_8_digital_outputs_O_186;
	::OutputVariables[5,187]	AT %QB."KUKA6_KRC5_ProfiNet_6_0".Module001_8_digital_outputs_O_187;
	::OutputVariables[5,188]	AT %QB."KUKA6_KRC5_ProfiNet_6_0".Module001_8_digital_outputs_O_188;
	::OutputVariables[5,189]	AT %QB."KUKA6_KRC5_ProfiNet_6_0".Module001_8_digital_outputs_O_189;
	::OutputVariables[5,190]	AT %QB."KUKA6_KRC5_ProfiNet_6_0".Module001_8_digital_outputs_O_190;
	::OutputVariables[5,191]	AT %QB."KUKA6_KRC5_ProfiNet_6_0".Module001_8_digital_outputs_O_191;
	::OutputVariables[5,192]	AT %QB."KUKA6_KRC5_ProfiNet_6_0".Module001_8_digital_outputs_O_192;
	::OutputVariables[5,193]	AT %QB."KUKA6_KRC5_ProfiNet_6_0".Module001_8_digital_outputs_O_193;
	::OutputVariables[5,194]	AT %QB."KUKA6_KRC5_ProfiNet_6_0".Module001_8_digital_outputs_O_194;
	::OutputVariables[5,195]	AT %QB."KUKA6_KRC5_ProfiNet_6_0".Module001_8_digital_outputs_O_195;
	::OutputVariables[5,196]	AT %QB."KUKA6_KRC5_ProfiNet_6_0".Module001_8_digital_outputs_O_196;
	::OutputVariables[5,197]	AT %QB."KUKA6_KRC5_ProfiNet_6_0".Module001_8_digital_outputs_O_197;
	::OutputVariables[5,198]	AT %QB."KUKA6_KRC5_ProfiNet_6_0".Module001_8_digital_outputs_O_198;
	::OutputVariables[5,199]	AT %QB."KUKA6_KRC5_ProfiNet_6_0".Module001_8_digital_outputs_O_199;
	::OutputVariables[5,200]	AT %QB."KUKA6_KRC5_ProfiNet_6_0".Module001_8_digital_outputs_O_200;
	::OutputVariables[5,201]	AT %QB."KUKA6_KRC5_ProfiNet_6_0".Module001_8_digital_outputs_O_201;
	::OutputVariables[5,202]	AT %QB."KUKA6_KRC5_ProfiNet_6_0".Module001_8_digital_outputs_O_202;
	::OutputVariables[5,203]	AT %QB."KUKA6_KRC5_ProfiNet_6_0".Module001_8_digital_outputs_O_203;
	::OutputVariables[5,204]	AT %QB."KUKA6_KRC5_ProfiNet_6_0".Module001_8_digital_outputs_O_204;
	::OutputVariables[5,205]	AT %QB."KUKA6_KRC5_ProfiNet_6_0".Module001_8_digital_outputs_O_205;
	::OutputVariables[5,206]	AT %QB."KUKA6_KRC5_ProfiNet_6_0".Module001_8_digital_outputs_O_206;
	::OutputVariables[5,207]	AT %QB."KUKA6_KRC5_ProfiNet_6_0".Module001_8_digital_outputs_O_207;
	::OutputVariables[5,208]	AT %QB."KUKA6_KRC5_ProfiNet_6_0".Module001_8_digital_outputs_O_208;
	::OutputVariables[5,209]	AT %QB."KUKA6_KRC5_ProfiNet_6_0".Module001_8_digital_outputs_O_209;
	::OutputVariables[5,210]	AT %QB."KUKA6_KRC5_ProfiNet_6_0".Module001_8_digital_outputs_O_210;
	::OutputVariables[5,211]	AT %QB."KUKA6_KRC5_ProfiNet_6_0".Module001_8_digital_outputs_O_211;
	::OutputVariables[5,212]	AT %QB."KUKA6_KRC5_ProfiNet_6_0".Module001_8_digital_outputs_O_212;
	::OutputVariables[5,213]	AT %QB."KUKA6_KRC5_ProfiNet_6_0".Module001_8_digital_outputs_O_213;
	::OutputVariables[5,214]	AT %QB."KUKA6_KRC5_ProfiNet_6_0".Module001_8_digital_outputs_O_214;
	::OutputVariables[5,215]	AT %QB."KUKA6_KRC5_ProfiNet_6_0".Module001_8_digital_outputs_O_215;
	::OutputVariables[5,216]	AT %QB."KUKA6_KRC5_ProfiNet_6_0".Module001_8_digital_outputs_O_216;
	::OutputVariables[5,217]	AT %QB."KUKA6_KRC5_ProfiNet_6_0".Module001_8_digital_outputs_O_217;
	::OutputVariables[5,218]	AT %QB."KUKA6_KRC5_ProfiNet_6_0".Module001_8_digital_outputs_O_218;
	::OutputVariables[5,219]	AT %QB."KUKA6_KRC5_ProfiNet_6_0".Module001_8_digital_outputs_O_219;
	::OutputVariables[5,220]	AT %QB."KUKA6_KRC5_ProfiNet_6_0".Module001_8_digital_outputs_O_220;
	::OutputVariables[5,221]	AT %QB."KUKA6_KRC5_ProfiNet_6_0".Module001_8_digital_outputs_O_221;
	::OutputVariables[5,222]	AT %QB."KUKA6_KRC5_ProfiNet_6_0".Module001_8_digital_outputs_O_222;
	::OutputVariables[5,223]	AT %QB."KUKA6_KRC5_ProfiNet_6_0".Module001_8_digital_outputs_O_223;
	::OutputVariables[5,224]	AT %QB."KUKA6_KRC5_ProfiNet_6_0".Module001_8_digital_outputs_O_224;
	::OutputVariables[5,225]	AT %QB."KUKA6_KRC5_ProfiNet_6_0".Module001_8_digital_outputs_O_225;
	::OutputVariables[5,226]	AT %QB."KUKA6_KRC5_ProfiNet_6_0".Module001_8_digital_outputs_O_226;
	::OutputVariables[5,227]	AT %QB."KUKA6_KRC5_ProfiNet_6_0".Module001_8_digital_outputs_O_227;
	::OutputVariables[5,228]	AT %QB."KUKA6_KRC5_ProfiNet_6_0".Module001_8_digital_outputs_O_228;
	::OutputVariables[5,229]	AT %QB."KUKA6_KRC5_ProfiNet_6_0".Module001_8_digital_outputs_O_229;
	::OutputVariables[5,230]	AT %QB."KUKA6_KRC5_ProfiNet_6_0".Module001_8_digital_outputs_O_230;
	::OutputVariables[5,231]	AT %QB."KUKA6_KRC5_ProfiNet_6_0".Module001_8_digital_outputs_O_231;
	::OutputVariables[5,232]	AT %QB."KUKA6_KRC5_ProfiNet_6_0".Module001_8_digital_outputs_O_232;
	::OutputVariables[5,233]	AT %QB."KUKA6_KRC5_ProfiNet_6_0".Module001_8_digital_outputs_O_233;
	::OutputVariables[5,234]	AT %QB."KUKA6_KRC5_ProfiNet_6_0".Module001_8_digital_outputs_O_234;
	::OutputVariables[5,235]	AT %QB."KUKA6_KRC5_ProfiNet_6_0".Module001_8_digital_outputs_O_235;
	::OutputVariables[5,236]	AT %QB."KUKA6_KRC5_ProfiNet_6_0".Module001_8_digital_outputs_O_236;
	::OutputVariables[5,237]	AT %QB."KUKA6_KRC5_ProfiNet_6_0".Module001_8_digital_outputs_O_237;
	::OutputVariables[5,238]	AT %QB."KUKA6_KRC5_ProfiNet_6_0".Module001_8_digital_outputs_O_238;
	::OutputVariables[5,239]	AT %QB."KUKA6_KRC5_ProfiNet_6_0".Module001_8_digital_outputs_O_239;
	::OutputVariables[5,240]	AT %QB."KUKA6_KRC5_ProfiNet_6_0".Module001_8_digital_outputs_O_240;
	::OutputVariables[5,241]	AT %QB."KUKA6_KRC5_ProfiNet_6_0".Module001_8_digital_outputs_O_241;
	::OutputVariables[5,242]	AT %QB."KUKA6_KRC5_ProfiNet_6_0".Module001_8_digital_outputs_O_242;
	::OutputVariables[5,243]	AT %QB."KUKA6_KRC5_ProfiNet_6_0".Module001_8_digital_outputs_O_243;
	::OutputVariables[5,244]	AT %QB."KUKA6_KRC5_ProfiNet_6_0".Module001_8_digital_outputs_O_244;
	::OutputVariables[5,245]	AT %QB."KUKA6_KRC5_ProfiNet_6_0".Module001_8_digital_outputs_O_245;
	::OutputVariables[5,246]	AT %QB."KUKA6_KRC5_ProfiNet_6_0".Module001_8_digital_outputs_O_246;
	::OutputVariables[5,247]	AT %QB."KUKA6_KRC5_ProfiNet_6_0".Module001_8_digital_outputs_O_247;
	::OutputVariables[5,248]	AT %QB."KUKA6_KRC5_ProfiNet_6_0".Module001_8_digital_outputs_O_248;
	::OutputVariables[5,249]	AT %QB."KUKA6_KRC5_ProfiNet_6_0".Module001_8_digital_outputs_O_249;
	::OutputVariables[5,250]	AT %QB."KUKA6_KRC5_ProfiNet_6_0".Module001_8_digital_outputs_O_250;
	::OutputVariables[5,251]	AT %QB."KUKA6_KRC5_ProfiNet_6_0".Module001_8_digital_outputs_O_251;
	::OutputVariables[5,252]	AT %QB."KUKA6_KRC5_ProfiNet_6_0".Module001_8_digital_outputs_O_252;
	::OutputVariables[5,253]	AT %QB."KUKA6_KRC5_ProfiNet_6_0".Module001_8_digital_outputs_O_253;

END_VAR
```

### PvMap.vvm - X20CP1685/PvMap.vvm
```iecst
VAR_CONFIG
	::Acopos6D:orderSpec AT %Q.::KUKA:orderSpec; (*Insert your comment here...*)
	::Acopos6D:orderAmount AT %Q.::KUKA:orderAmount; (*Insert your comment here...*)
	::Acopos6D:robotExecute AT %Q.::KUKA:robotExecute; (*Insert your comment here...*)
	::KUKA:robotBusy AT %Q.::Acopos6D:robotBusy; (*Insert your comment here...*)
	::KUKA:robotDone AT %Q.::Acopos6D:robotDone; (*Insert your comment here...*)
END_VAR
```
